LIN {X 0,Y 210.301,Z 279.738,A -85,B 0,C 180,E1 -24809.445,E2 -24809.445} C_VEL
LIN {X 0,Y 205.69,Z 270.017,A -85,B 0,C 180,E1 -24812.462,E2 -24812.462} C_VEL
LIN {X 0,Y 202.047,Z 263.223,A -85,B 0,C 180,E1 -24815.123,E2 -24815.123} C_VEL
LIN {X 0,Y 198.531,Z 257.151,A -85,B 0,C 180,E1 -24818.043,E2 -24818.043} C_VEL
LIN {X 0,Y 194.726,Z 251.083,A -85,B 0,C 180,E1 -24821.795,E2 -24821.795} C_VEL
LIN {X 0,Y 192.117,Z 247.147,A -85,B 0,C 180,E1 -24824.974,E2 -24824.974} C_VEL
LIN {X 0,Y 189.866,Z 243.661,A -85,B 0,C 180,E1 -24828.524,E2 -24828.524} C_VEL
LIN {X 0,Y 187.215,Z 239.674,A -85,B 0,C 180,E1 -24835.964,E2 -24835.964} C_VEL
LIN {X 0,Y 187.003,Z 239.077,A -85,B 0,C 180,E1 -24837.846,E2 -24837.846} C_VEL
LIN {X 0,Y 186.955,Z 239.01,A -85,B 0,C 180,E1 -24840.538,E2 -24840.538} C_VEL
LIN {X 0,Y 188.211,Z 242.32,A -85,B 0,C 180,E1 -24847.24,E2 -24847.24} C_VEL
LIN {X 0,Y 189.577,Z 244.391,A -85,B 0,C 180,E1 -24850.277,E2 -24850.277} C_VEL
LIN {X 0,Y 192.089,Z 248.48,A -85,B 0,C 180,E1 -24854.298,E2 -24854.298} C_VEL
LIN {X 0,Y 195.023,Z 253.243,A -85,B 0,C 180,E1 -24857.837,E2 -24857.837} C_VEL
LIN {X 0,Y 198.75,Z 259.543,A -85,B 0,C 180,E1 -24861.454,E2 -24861.454} C_VEL
LIN {X 0,Y 202.456,Z 266.139,A -85,B 0,C 180,E1 -24864.481,E2 -24864.481} C_VEL
LIN {X 0,Y 205.633,Z 272.337,A -85,B 0,C 180,E1 -24866.789,E2 -24866.789} C_VEL
LIN {X 0,Y 208.488,Z 283.961,A -85,B 0,C 180,E1 -24869.081,E2 -24869.081} C_VEL
LIN {X 0,Y 208.34,Z 300.022,A -85,B 0,C 180,E1 -24870.092,E2 -24870.092} C_VEL
LIN {X 0,Y 201.69,Z 376.905,A -85,B 0,C 180,E1 -24872.216,E2 -24872.216} C_VEL
LIN {X 0,Y 199.026,Z 392.933,A -85,B 0,C 180,E1 -24872.89,E2 -24872.89} C_VEL
LIN {X 0,Y 195.992,Z 405.457,A -85,B 0,C 180,E1 -24873.625,E2 -24873.625} C_VEL
LIN {X 0,Y 194.072,Z 410.997,A -85,B 0,C 180,E1 -24873.869,E2 -24873.869} C_VEL
LIN {X 0,Y 189.476,Z 419.824,A -85,B 0,C 180,E1 -24873.895,E2 -24873.895} C_VEL
LIN {X 0,Y 184.541,Z 428.454,A -85,B 0,C 180,E1 -24874.027,E2 -24874.027} C_VEL
LIN {X 0,Y 182.039,Z 433.552,A -85,B 0,C 180,E1 -24874.466,E2 -24874.466} C_VEL
LIN {X 0,Y 176.253,Z 445.926,A -85,B 0,C 180,E1 -24876.157,E2 -24876.157} C_VEL
LIN {X 0,Y 169.53,Z 458.558,A -85,B 0,C 180,E1 -24878.45,E2 -24878.45} C_VEL
LIN {X 0,Y 162.971,Z 469.426,A -85,B 0,C 180,E1 -24881.009,E2 -24881.009} C_VEL
LIN {X 0,Y 156.265,Z 479.356,A -85,B 0,C 180,E1 -24883.984,E2 -24883.984} C_VEL
LIN {X 0,Y 149.299,Z 489.115,A -85,B 0,C 180,E1 -24887.877,E2 -24887.877} C_VEL
LIN {X 0,Y 143.262,Z 496.88,A -85,B 0,C 180,E1 -24891.86,E2 -24891.86} C_VEL
LIN {X 0,Y 138.473,Z 503.139,A -85,B 0,C 180,E1 -24896.067,E2 -24896.067} C_VEL
LIN {X 0,Y 133.419,Z 509.601,A -85,B 0,C 180,E1 -24901.705,E2 -24901.705} C_VEL
LIN {X 0,Y 129.8,Z 514.638,A -85,B 0,C 180,E1 -24907.732,E2 -24907.732} C_VEL
LIN {X 0,Y 127.56,Z 518.367,A -85,B 0,C 180,E1 -24914.014,E2 -24914.014} C_VEL
LIN {X 0,Y 126.835,Z 520.883,A -85,B 0,C 180,E1 -24920.435,E2 -24920.435} C_VEL
LIN {X 0,Y 127.101,Z 521.841,A -85,B 0,C 180,E1 -24924.439,E2 -24924.439} C_VEL
LIN {X 0,Y 127.589,Z 522.401,A -85,B 0,C 180,E1 -24930.004,E2 -24930.004} C_VEL
LIN {X 0,Y 127.142,Z 521.8,A -85,B 0,C 180,E1 -24935.747,E2 -24935.747} C_VEL
LIN {X 0,Y 127.052,Z 519.741,A -85,B 0,C 180,E1 -24942.787,E2 -24942.787} C_VEL
LIN {X 0,Y 128.532,Z 516.599,A -85,B 0,C 180,E1 -24949.156,E2 -24949.156} C_VEL
LIN {X 0,Y 131.403,Z 512.192,A -85,B 0,C 180,E1 -24955.337,E2 -24955.337} C_VEL
LIN {X 0,Y 135.799,Z 506.44,A -85,B 0,C 180,E1 -24961.171,E2 -24961.171} C_VEL
LIN {X 0,Y 141.47,Z 499.175,A -85,B 0,C 180,E1 -24966.598,E2 -24966.598} C_VEL
LIN {X 0,Y 146.575,Z 492.646,A -85,B 0,C 180,E1 -24970.343,E2 -24970.343} C_VEL
LIN {X 0,Y 152.637,Z 485.303,A -85,B 0,C 180,E1 -24973.573,E2 -24973.573} C_VEL
LIN {X 0,Y 161.541,Z 483.741,A -85,B 0,C 180,E1 -24977.702,E2 -24977.702} C_VEL
LIN {X 0,Y 172.128,Z 481.337,A -85,B 0,C 180,E1 -24981.424,E2 -24981.424} C_VEL
LIN {X 0,Y 171.753,Z 480.963,A -85,B 0,C 180,E1 -24982.136,E2 -24982.136} C_VEL
LIN {X 0,Y 162.139,Z 479.16,A -85,B 0,C 180,E1 -24985.703,E2 -24985.703} C_VEL
LIN {X 0,Y 153.483,Z 476.191,A -85,B 0,C 180,E1 -24989.756,E2 -24989.756} C_VEL
LIN {X 0,Y 145.911,Z 472.001,A -85,B 0,C 180,E1 -24994.311,E2 -24994.311} C_VEL
LIN {X 0,Y 139.663,Z 466.519,A -85,B 0,C 180,E1 -24999.375,E2 -24999.375} C_VEL
LIN {X 0,Y 135.041,Z 459.696,A -85,B 0,C 180,E1 -25004.917,E2 -25004.917} C_VEL
LIN {X 0,Y 132.875,Z 454.923,A -85,B 0,C 180,E1 -25008.367,E2 -25008.367} C_VEL
LIN {X 0,Y 131.811,Z 454.489,A -85,B 0,C 180,E1 -25010.796,E2 -25010.796} C_VEL
LIN {X 0,Y 132.801,Z 449.564,A -85,B 0,C 180,E1 -25020,E2 -25020} C_VEL
LIN {X 0,Y 134.381,Z 447.309,A -85,B 0,C 180,E1 -25022.998,E2 -25022.998} C_VEL
LIN {X 0,Y 136.769,Z 444.692,A -85,B 0,C 180,E1 -25027.381,E2 -25027.381} C_VEL
LIN {X 0,Y 140.175,Z 441.466,A -85,B 0,C 180,E1 -25031.264,E2 -25031.264} C_VEL
LIN {X 0,Y 143.118,Z 439.169,A -85,B 0,C 180,E1 -25034.214,E2 -25034.214} C_VEL
LIN {X 0,Y 146.772,Z 436.106,A -85,B 0,C 180,E1 -25036.697,E2 -25036.697} C_VEL
LIN {X 0,Y 151.382,Z 432.821,A -85,B 0,C 180,E1 -25039.924,E2 -25039.924} C_VEL
LIN {X 0,Y 156.65,Z 428.519,A -85,B 0,C 180,E1 -25042.417,E2 -25042.417} C_VEL
LIN {X 0,Y 160.693,Z 425.786,A -85,B 0,C 180,E1 -25044.55,E2 -25044.55} C_VEL
LIN {X 0,Y 167.067,Z 420.351,A -85,B 0,C 180,E1 -25046.819,E2 -25046.819} C_VEL
LIN {X 0,Y 170.649,Z 417.188,A -85,B 0,C 180,E1 -25048.005,E2 -25048.005} C_VEL
LIN {X 0,Y 176.406,Z 412.41,A -85,B 0,C 180,E1 -25049.868,E2 -25049.868} C_VEL
LIN {X 0,Y 182.287,Z 406.571,A -85,B 0,C 180,E1 -25051.364,E2 -25051.364} C_VEL
LIN {X 0,Y 188.257,Z 399.411,A -85,B 0,C 180,E1 -25052.536,E2 -25052.536} C_VEL
LIN {X 0,Y 191.638,Z 395.946,A -85,B 0,C 180,E1 -25053.374,E2 -25053.374} C_VEL
LIN {X 0,Y 191.708,Z 397.569,A -85,B 0,C 180,E1 -25053.78,E2 -25053.78} C_VEL
LIN {X 0,Y 187.24,Z 410.98,A -85,B 0,C 180,E1 -25055.272,E2 -25055.272} C_VEL
LIN {X 0,Y 181.776,Z 424.211,A -85,B 0,C 180,E1 -25057.111,E2 -25057.111} C_VEL
LIN {X 0,Y 175.849,Z 436.31,A -85,B 0,C 180,E1 -25059.251,E2 -25059.251} C_VEL
LIN {X 0,Y 169.638,Z 447.434,A -85,B 0,C 180,E1 -25061.774,E2 -25061.774} C_VEL
LIN {X 0,Y 163.383,Z 457.621,A -85,B 0,C 180,E1 -25064.781,E2 -25064.781} C_VEL
LIN {X 0,Y 156.338,Z 467.581,A -85,B 0,C 180,E1 -25068.462,E2 -25068.462} C_VEL
LIN {X 0,Y 149.927,Z 475.829,A -85,B 0,C 180,E1 -25072.451,E2 -25072.451} C_VEL
LIN {X 0,Y 143.625,Z 483.517,A -85,B 0,C 180,E1 -25077.431,E2 -25077.431} C_VEL
LIN {X 0,Y 138.146,Z 489.63,A -85,B 0,C 180,E1 -25082.747,E2 -25082.747} C_VEL
LIN {X 0,Y 133.9,Z 494.331,A -85,B 0,C 180,E1 -25088.44,E2 -25088.44} C_VEL
LIN {X 0,Y 130.785,Z 497.762,A -85,B 0,C 180,E1 -25094.41,E2 -25094.41} C_VEL
LIN {X 0,Y 128.776,Z 500.015,A -85,B 0,C 180,E1 -25100.573,E2 -25100.573} C_VEL
LIN {X 0,Y 127.806,Z 501.153,A -85,B 0,C 180,E1 -25106.844,E2 -25106.844} C_VEL
LIN {X 0,Y 127.802,Z 501.162,A -85,B 0,C 180,E1 -25113.148,E2 -25113.148} C_VEL
LIN {X 0,Y 128.768,Z 500.062,A -85,B 0,C 180,E1 -25119.42,E2 -25119.42} C_VEL
LIN {X 0,Y 130.775,Z 497.85,A -85,B 0,C 180,E1 -25125.583,E2 -25125.583} C_VEL
LIN {X 0,Y 133.858,Z 494.47,A -85,B 0,C 180,E1 -25131.559,E2 -25131.559} C_VEL
LIN {X 0,Y 138.082,Z 489.818,A -85,B 0,C 180,E1 -25137.258,E2 -25137.258} C_VEL
LIN {X 0,Y 143.533,Z 483.748,A -85,B 0,C 180,E1 -25142.584,E2 -25142.584} C_VEL
LIN {X 0,Y 149.833,Z 476.111,A -85,B 0,C 180,E1 -25147.568,E2 -25147.568} C_VEL
LIN {X 0,Y 156.244,Z 467.927,A -85,B 0,C 180,E1 -25151.56,E2 -25151.56} C_VEL
LIN {X 0,Y 163.227,Z 458.042,A -85,B 0,C 180,E1 -25155.265,E2 -25155.265} C_VEL
LIN {X 0,Y 169.531,Z 447.93,A -85,B 0,C 180,E1 -25158.257,E2 -25158.257} C_VEL
LIN {X 0,Y 175.806,Z 436.902,A -85,B 0,C 180,E1 -25160.757,E2 -25160.757} C_VEL
LIN {X 0,Y 181.69,Z 424.906,A -85,B 0,C 180,E1 -25162.915,E2 -25162.915} C_VEL
LIN {X 0,Y 187.164,Z 411.807,A -85,B 0,C 180,E1 -25164.752,E2 -25164.752} C_VEL
LIN {X 0,Y 191.739,Z 398.192,A -85,B 0,C 180,E1 -25166.288,E2 -25166.288} C_VEL
LIN {X 0,Y 195.352,Z 384.362,A -85,B 0,C 180,E1 -25167.521,E2 -25167.521} C_VEL
LIN {X 0,Y 198.346,Z 369.373,A -85,B 0,C 180,E1 -25168.468,E2 -25168.468} C_VEL
LIN {X 0,Y 200.316,Z 354.638,A -85,B 0,C 180,E1 -25169.082,E2 -25169.082} C_VEL
LIN {X 0,Y 206.565,Z 283.097,A -85,B 0,C 180,E1 -25171.043,E2 -25171.043} C_VEL
LIN {X 0,Y 202.838,Z 275.011,A -85,B 0,C 180,E1 -25173.681,E2 -25173.681} C_VEL
LIN {X 0,Y 199.598,Z 268.732,A -85,B 0,C 180,E1 -25176.224,E2 -25176.224} C_VEL
LIN {X 0,Y 196.564,Z 263.306,A -85,B 0,C 180,E1 -25178.913,E2 -25178.913} C_VEL
LIN {X 0,Y 193.052,Z 257.443,A -85,B 0,C 180,E1 -25182.603,E2 -25182.603} C_VEL
LIN {X 0,Y 190.738,Z 253.83,A -85,B 0,C 180,E1 -25185.598,E2 -25185.598} C_VEL
LIN {X 0,Y 188.711,Z 250.517,A -85,B 0,C 180,E1 -25188.996,E2 -25188.996} C_VEL
LIN {X 0,Y 186.324,Z 246.732,A -85,B 0,C 180,E1 -25196.08,E2 -25196.08} C_VEL
LIN {X 0,Y 186.138,Z 246.132,A -85,B 0,C 180,E1 -25197.836,E2 -25197.836} C_VEL
LIN {X 0,Y 186.09,Z 246.061,A -85,B 0,C 180,E1 -25200.541,E2 -25200.541} C_VEL
LIN {X 0,Y 188.131,Z 250.58,A -85,B 0,C 180,E1 -25209.135,E2 -25209.135} C_VEL
LIN {X 0,Y 190.741,Z 255.196,A -85,B 0,C 180,E1 -25213.721,E2 -25213.721} C_VEL
LIN {X 0,Y 193.391,Z 259.687,A -85,B 0,C 180,E1 -25217.105,E2 -25217.105} C_VEL
LIN {X 0,Y 196.826,Z 265.796,A -85,B 0,C 180,E1 -25220.646,E2 -25220.646} C_VEL
LIN {X 0,Y 200.257,Z 272.156,A -85,B 0,C 180,E1 -25223.614,E2 -25223.614} C_VEL
LIN {X 0,Y 202.814,Z 277.371,A -85,B 0,C 180,E1 -25225.599,E2 -25225.599} C_VEL
LIN {X 0,Y 204.982,Z 286.69,A -85,B 0,C 180,E1 -25227.502,E2 -25227.502} C_VEL
LIN {X 0,Y 204.794,Z 300.471,A -85,B 0,C 180,E1 -25228.399,E2 -25228.399} C_VEL
LIN {X 0,Y 197.965,Z 376.592,A -85,B 0,C 180,E1 -25230.478,E2 -25230.478} C_VEL
LIN {X 0,Y 195.405,Z 391.525,A -85,B 0,C 180,E1 -25231.086,E2 -25231.086} C_VEL
LIN {X 0,Y 191.613,Z 406.898,A -85,B 0,C 180,E1 -25231.992,E2 -25231.992} C_VEL
LIN {X 0,Y 186.835,Z 421.579,A -85,B 0,C 180,E1 -25233.185,E2 -25233.185} C_VEL
LIN {X 0,Y 182.039,Z 433.552,A -85,B 0,C 180,E1 -25234.466,E2 -25234.466} C_VEL
LIN {X 0,Y 180.165,Z 436.986,A -85,B 0,C 180,E1 -25234.726,E2 -25234.726} C_VEL
LIN {X 0,Y 175.915,Z 442.251,A -85,B 0,C 180,E1 -25234.698,E2 -25234.698} C_VEL
LIN {X 0,Y 171.494,Z 447.391,A -85,B 0,C 180,E1 -25234.721,E2 -25234.721} C_VEL
LIN {X 0,Y 169.356,Z 450.558,A -85,B 0,C 180,E1 -25235.084,E2 -25235.084} C_VEL
LIN {X 0,Y 162.542,Z 462.474,A -85,B 0,C 180,E1 -25237.515,E2 -25237.515} C_VEL
LIN {X 0,Y 156.017,Z 472.377,A -85,B 0,C 180,E1 -25240.028,E2 -25240.028} C_VEL
LIN {X 0,Y 149.199,Z 481.767,A -85,B 0,C 180,E1 -25243.109,E2 -25243.109} C_VEL
LIN {X 0,Y 142.066,Z 491.018,A -85,B 0,C 180,E1 -25247.145,E2 -25247.145} C_VEL
LIN {X 0,Y 135.713,Z 498.723,A -85,B 0,C 180,E1 -25251.585,E2 -25251.585} C_VEL
LIN {X 0,Y 129.645,Z 505.962,A -85,B 0,C 180,E1 -25257.179,E2 -25257.179} C_VEL
LIN {X 0,Y 124.93,Z 511.693,A -85,B 0,C 180,E1 -25263.258,E2 -25263.258} C_VEL
LIN {X 0,Y 121.736,Z 516.066,A -85,B 0,C 180,E1 -25269.738,E2 -25269.738} C_VEL
LIN {X 0,Y 120.018,Z 519.18,A -85,B 0,C 180,E1 -25276.458,E2 -25276.458} C_VEL
LIN {X 0,Y 119.884,Z 521.109,A -85,B 0,C 180,E1 -25283.271,E2 -25283.271} C_VEL
LIN {X 0,Y 120.207,Z 521.624,A -85,B 0,C 180,E1 -25286.653,E2 -25286.653} C_VEL
LIN {X 0,Y 120.5,Z 521.815,A -85,B 0,C 180,E1 -25290.004,E2 -25290.004} C_VEL
LIN {X 0,Y 120.06,Z 521.279,A -85,B 0,C 180,E1 -25295.657,E2 -25295.657} C_VEL
LIN {X 0,Y 119.81,Z 520.269,A -85,B 0,C 180,E1 -25300.14,E2 -25300.14} C_VEL
LIN {X 0,Y 120.683,Z 517.725,A -85,B 0,C 180,E1 -25306.933,E2 -25306.933} C_VEL
LIN {X 0,Y 123.126,Z 513.96,A -85,B 0,C 180,E1 -25313.555,E2 -25313.555} C_VEL
LIN {X 0,Y 127.128,Z 508.897,A -85,B 0,C 180,E1 -25319.842,E2 -25319.842} C_VEL
LIN {X 0,Y 132.577,Z 502.415,A -85,B 0,C 180,E1 -25325.675,E2 -25325.675} C_VEL
LIN {X 0,Y 138.153,Z 495.656,A -85,B 0,C 180,E1 -25330.265,E2 -25330.265} C_VEL
LIN {X 0,Y 145.433,Z 487.123,A -85,B 0,C 180,E1 -25334.488,E2 -25334.488} C_VEL
LIN {X 0,Y 148.59,Z 483.626,A -85,B 0,C 180,E1 -25335.922,E2 -25335.922} C_VEL
LIN {X 0,Y 161.85,Z 481.639,A -85,B 0,C 180,E1 -25341.413,E2 -25341.413} C_VEL
LIN {X 0,Y 161.175,Z 481.066,A -85,B 0,C 180,E1 -25342.377,E2 -25342.377} C_VEL
LIN {X 0,Y 151.756,Z 478.235,A -85,B 0,C 180,E1 -25346.239,E2 -25346.239} C_VEL
LIN {X 0,Y 143.269,Z 474.219,A -85,B 0,C 180,E1 -25350.624,E2 -25350.624} C_VEL
LIN {X 0,Y 136.177,Z 468.955,A -85,B 0,C 180,E1 -25355.615,E2 -25355.615} C_VEL
LIN {X 0,Y 131.032,Z 463.521,A -85,B 0,C 180,E1 -25360.414,E2 -25360.414} C_VEL
LIN {X 0,Y 128.644,Z 462.497,A -85,B 0,C 180,E1 -25364.148,E2 -25364.148} C_VEL
LIN {X 0,Y 127.926,Z 460.868,A -85,B 0,C 180,E1 -25367.306,E2 -25367.306} C_VEL
LIN {X 0,Y 127.086,Z 459.748,A -85,B 0,C 180,E1 -25370.451,E2 -25370.451} C_VEL
LIN {X 0,Y 128.034,Z 455.043,A -85,B 0,C 180,E1 -25380,E2 -25380} C_VEL
LIN {X 0,Y 133.201,Z 449.373,A -85,B 0,C 180,E1 -25389.108,E2 -25389.108} C_VEL
LIN {X 0,Y 135.913,Z 447.051,A -85,B 0,C 180,E1 -25391.937,E2 -25391.937} C_VEL
LIN {X 0,Y 140.264,Z 443.953,A -85,B 0,C 180,E1 -25395.997,E2 -25395.997} C_VEL
LIN {X 0,Y 143.533,Z 441.403,A -85,B 0,C 180,E1 -25398.062,E2 -25398.062} C_VEL
LIN {X 0,Y 147.722,Z 438.705,A -85,B 0,C 180,E1 -25400.905,E2 -25400.905} C_VEL
LIN {X 0,Y 153.368,Z 434.562,A -85,B 0,C 180,E1 -25403.575,E2 -25403.575} C_VEL
LIN {X 0,Y 154.685,Z 433.547,A -85,B 0,C 180,E1 -25404.137,E2 -25404.137} C_VEL
LIN {X 0,Y 159.011,Z 430.838,A -85,B 0,C 180,E1 -25406.231,E2 -25406.231} C_VEL
LIN {X 0,Y 165.803,Z 425.469,A -85,B 0,C 180,E1 -25408.482,E2 -25408.482} C_VEL
LIN {X 0,Y 170.018,Z 422.026,A -85,B 0,C 180,E1 -25409.739,E2 -25409.739} C_VEL
LIN {X 0,Y 176.299,Z 417.087,A -85,B 0,C 180,E1 -25411.598,E2 -25411.598} C_VEL
LIN {X 0,Y 183.059,Z 410.79,A -85,B 0,C 180,E1 -25413.132,E2 -25413.132} C_VEL
LIN {X 0,Y 182.832,Z 412.616,A -85,B 0,C 180,E1 -25413.597,E2 -25413.597} C_VEL
LIN {X 0,Y 176.996,Z 426.093,A -85,B 0,C 180,E1 -25415.508,E2 -25415.508} C_VEL
LIN {X 0,Y 170.881,Z 438.007,A -85,B 0,C 180,E1 -25417.65,E2 -25417.65} C_VEL
LIN {X 0,Y 163.864,Z 449.871,A -85,B 0,C 180,E1 -25420.418,E2 -25420.418} C_VEL
LIN {X 0,Y 157.419,Z 459.784,A -85,B 0,C 180,E1 -25423.487,E2 -25423.487} C_VEL
LIN {X 0,Y 150.117,Z 469.477,A -85,B 0,C 180,E1 -25427.243,E2 -25427.243} C_VEL
LIN {X 0,Y 143.171,Z 477.858,A -85,B 0,C 180,E1 -25431.55,E2 -25431.55} C_VEL
LIN {X 0,Y 137.709,Z 484.102,A -85,B 0,C 180,E1 -25435.844,E2 -25435.844} C_VEL
LIN {X 0,Y 131.884,Z 490.216,A -85,B 0,C 180,E1 -25441.336,E2 -25441.336} C_VEL
LIN {X 0,Y 127.339,Z 494.916,A -85,B 0,C 180,E1 -25447.269,E2 -25447.269} C_VEL
LIN {X 0,Y 123.964,Z 498.349,A -85,B 0,C 180,E1 -25453.528,E2 -25453.528} C_VEL
LIN {X 0,Y 121.814,Z 500.599,A -85,B 0,C 180,E1 -25460.029,E2 -25460.029} C_VEL
LIN {X 0,Y 120.741,Z 501.738,A -85,B 0,C 180,E1 -25466.659,E2 -25466.659} C_VEL
LIN {X 0,Y 120.737,Z 501.747,A -85,B 0,C 180,E1 -25473.333,E2 -25473.333} C_VEL
LIN {X 0,Y 121.806,Z 500.645,A -85,B 0,C 180,E1 -25479.963,E2 -25479.963} C_VEL
LIN {X 0,Y 123.953,Z 498.436,A -85,B 0,C 180,E1 -25486.464,E2 -25486.464} C_VEL
LIN {X 0,Y 127.3,Z 495.053,A -85,B 0,C 180,E1 -25492.73,E2 -25492.73} C_VEL
LIN {X 0,Y 131.825,Z 490.401,A -85,B 0,C 180,E1 -25498.669,E2 -25498.669} C_VEL
LIN {X 0,Y 137.596,Z 484.332,A -85,B 0,C 180,E1 -25504.179,E2 -25504.179} C_VEL
LIN {X 0,Y 144.282,Z 476.693,A -85,B 0,C 180,E1 -25509.284,E2 -25509.284} C_VEL
LIN {X 0,Y 151.006,Z 468.508,A -85,B 0,C 180,E1 -25513.347,E2 -25513.347} C_VEL
LIN {X 0,Y 157.28,Z 460.181,A -85,B 0,C 180,E1 -25516.557,E2 -25516.557} C_VEL
LIN {X 0,Y 163.766,Z 450.319,A -85,B 0,C 180,E1 -25519.612,E2 -25519.612} C_VEL
LIN {X 0,Y 170.814,Z 438.546,A -85,B 0,C 180,E1 -25522.37,E2 -25522.37} C_VEL
LIN {X 0,Y 176.914,Z 426.736,A -85,B 0,C 180,E1 -25524.52,E2 -25524.52} C_VEL
LIN {X 0,Y 181.91,Z 415.45,A -85,B 0,C 180,E1 -25526.159,E2 -25526.159} C_VEL
LIN {X 0,Y 186.691,Z 402.462,A -85,B 0,C 180,E1 -25527.697,E2 -25527.697} C_VEL
LIN {X 0,Y 190.649,Z 388.919,A -85,B 0,C 180,E1 -25528.982,E2 -25528.982} C_VEL
LIN {X 0,Y 193.969,Z 374.104,A -85,B 0,C 180,E1 -25530.012,E2 -25530.012} C_VEL
LIN {X 0,Y 196.25,Z 359.84,A -85,B 0,C 180,E1 -25530.679,E2 -25530.679} C_VEL
LIN {X 0,Y 199.856,Z 320.402,A -85,B 0,C 180,E1 -25531.84,E2 -25531.84} C_VEL
LIN {X 0,Y 202.956,Z 286.419,A -85,B 0,C 180,E1 -25532.723,E2 -25532.723} C_VEL
LIN {X 0,Y 199.718,Z 279.221,A -85,B 0,C 180,E1 -25535.23,E2 -25535.23} C_VEL
LIN {X 0,Y 196.437,Z 272.696,A -85,B 0,C 180,E1 -25538.073,E2 -25538.073} C_VEL
LIN {X 0,Y 193.332,Z 267.144,A -85,B 0,C 180,E1 -25541.178,E2 -25541.178} C_VEL
LIN {X 0,Y 191.177,Z 263.47,A -85,B 0,C 180,E1 -25543.721,E2 -25543.721} C_VEL
LIN {X 0,Y 189.421,Z 260.538,A -85,B 0,C 180,E1 -25546.181,E2 -25546.181} C_VEL
LIN {X 0,Y 187.57,Z 257.366,A -85,B 0,C 180,E1 -25549.475,E2 -25549.475} C_VEL
LIN {X 0,Y 185.347,Z 253.38,A -85,B 0,C 180,E1 -25557.011,E2 -25557.011} C_VEL
LIN {X 0,Y 185.223,Z 253.121,A -85,B 0,C 180,E1 -25560.543,E2 -25560.543} C_VEL
LIN {X 0,Y 187.07,Z 257.557,A -85,B 0,C 180,E1 -25568.779,E2 -25568.779} C_VEL
LIN {X 0,Y 189.332,Z 261.737,A -85,B 0,C 180,E1 -25573.005,E2 -25573.005} C_VEL
LIN {X 0,Y 191.838,Z 266.266,A -85,B 0,C 180,E1 -25576.426,E2 -25576.426} C_VEL
LIN {X 0,Y 194.952,Z 272.062,A -85,B 0,C 180,E1 -25579.831,E2 -25579.831} C_VEL
LIN {X 0,Y 198.041,Z 278.053,A -85,B 0,C 180,E1 -25582.673,E2 -25582.673} C_VEL
LIN {X 0,Y 200.081,Z 282.443,A -85,B 0,C 180,E1 -25584.376,E2 -25584.376} C_VEL
LIN {X 0,Y 201.578,Z 289.429,A -85,B 0,C 180,E1 -25585.837,E2 -25585.837} C_VEL
LIN {X 0,Y 201.377,Z 301.467,A -85,B 0,C 180,E1 -25586.658,E2 -25586.658} C_VEL
LIN {X 0,Y 194.542,Z 375.348,A -85,B 0,C 180,E1 -25588.648,E2 -25588.648} C_VEL
LIN {X 0,Y 192.015,Z 390.106,A -85,B 0,C 180,E1 -25589.231,E2 -25589.231} C_VEL
LIN {X 0,Y 188.294,Z 405.073,A -85,B 0,C 180,E1 -25590.071,E2 -25590.071} C_VEL
LIN {X 0,Y 183.734,Z 419.063,A -85,B 0,C 180,E1 -25591.151,E2 -25591.151} C_VEL
LIN {X 0,Y 178.2,Z 432.753,A -85,B 0,C 180,E1 -25592.547,E2 -25592.547} C_VEL
LIN {X 0,Y 172.136,Z 445.352,A -85,B 0,C 180,E1 -25594.238,E2 -25594.238} C_VEL
LIN {X 0,Y 169.356,Z 450.558,A -85,B 0,C 180,E1 -25595.084,E2 -25595.084} C_VEL
LIN {X 0,Y 166.353,Z 455.267,A -85,B 0,C 180,E1 -25595.783,E2 -25595.783} C_VEL
LIN {X 0,Y 160.083,Z 462.596,A -85,B 0,C 180,E1 -25596.579,E2 -25596.579} C_VEL
LIN {X 0,Y 153.536,Z 469.587,A -85,B 0,C 180,E1 -25597.532,E2 -25597.532} C_VEL
LIN {X 0,Y 150.13,Z 473.642,A -85,B 0,C 180,E1 -25598.509,E2 -25598.509} C_VEL
LIN {X 0,Y 143.287,Z 482.598,A -85,B 0,C 180,E1 -25601.59,E2 -25601.59} C_VEL
LIN {X 0,Y 135.88,Z 491.624,A -85,B 0,C 180,E1 -25605.719,E2 -25605.719} C_VEL
LIN {X 0,Y 130.108,Z 498.128,A -85,B 0,C 180,E1 -25609.6,E2 -25609.6} C_VEL
LIN {X 0,Y 123.647,Z 505.369,A -85,B 0,C 180,E1 -25615.367,E2 -25615.367} C_VEL
LIN {X 0,Y 118.533,Z 511.099,A -85,B 0,C 180,E1 -25621.689,E2 -25621.689} C_VEL
LIN {X 0,Y 114.999,Z 515.471,A -85,B 0,C 180,E1 -25628.494,E2 -25628.494} C_VEL
LIN {X 0,Y 113.05,Z 518.587,A -85,B 0,C 180,E1 -25635.606,E2 -25635.606} C_VEL
LIN {X 0,Y 112.761,Z 520.516,A -85,B 0,C 180,E1 -25642.844,E2 -25642.844} C_VEL
LIN {X 0,Y 113.097,Z 521.035,A -85,B 0,C 180,E1 -25646.442,E2 -25646.442} C_VEL
LIN {X 0,Y 113.414,Z 521.229,A -85,B 0,C 180,E1 -25650.005,E2 -25650.005} C_VEL
LIN {X 0,Y 112.988,Z 520.752,A -85,B 0,C 180,E1 -25655.605,E2 -25655.605} C_VEL
LIN {X 0,Y 112.735,Z 519.674,A -85,B 0,C 180,E1 -25660.784,E2 -25660.784} C_VEL
LIN {X 0,Y 113.822,Z 517.131,A -85,B 0,C 180,E1 -25667.987,E2 -25667.987} C_VEL
LIN {X 0,Y 116.86,Z 512.975,A -85,B 0,C 180,E1 -25675.565,E2 -25675.565} C_VEL
LIN {X 0,Y 120.938,Z 508.302,A -85,B 0,C 180,E1 -25681.539,E2 -25681.539} C_VEL
LIN {X 0,Y 126.797,Z 501.82,A -85,B 0,C 180,E1 -25687.572,E2 -25687.572} C_VEL
LIN {X 0,Y 132.195,Z 495.676,A -85,B 0,C 180,E1 -25691.902,E2 -25691.902} C_VEL
LIN {X 0,Y 139.29,Z 487.783,A -85,B 0,C 180,E1 -25695.976,E2 -25695.976} C_VEL
LIN {X 0,Y 144.835,Z 481.78,A -85,B 0,C 180,E1 -25698.385,E2 -25698.385} C_VEL
LIN {X 0,Y 152.452,Z 481.01,A -85,B 0,C 180,E1 -25701.605,E2 -25701.605} C_VEL
LIN {X 0,Y 150.629,Z 480.237,A -85,B 0,C 180,E1 -25702.66,E2 -25702.66} C_VEL
LIN {X 0,Y 141.375,Z 476.387,A -85,B 0,C 180,E1 -25706.851,E2 -25706.851} C_VEL
LIN {X 0,Y 132.785,Z 471.077,A -85,B 0,C 180,E1 -25711.983,E2 -25711.983} C_VEL
LIN {X 0,Y 129.929,Z 470.653,A -85,B 0,C 180,E1 -25714.36,E2 -25714.36} C_VEL
LIN {X 0,Y 127.417,Z 469.706,A -85,B 0,C 180,E1 -25717.288,E2 -25717.288} C_VEL
LIN {X 0,Y 125.607,Z 468.411,A -85,B 0,C 180,E1 -25720.384,E2 -25720.384} C_VEL
LIN {X 0,Y 123.763,Z 467.51,A -85,B 0,C 180,E1 -25723.505,E2 -25723.505} C_VEL
LIN {X 0,Y 121.853,Z 463.487,A -85,B 0,C 180,E1 -25733.376,E2 -25733.376} C_VEL
LIN {X 0,Y 124.383,Z 458.597,A -85,B 0,C 180,E1 -25743.239,E2 -25743.239} C_VEL
LIN {X 0,Y 129.591,Z 453.901,A -85,B 0,C 180,E1 -25750.942,E2 -25750.942} C_VEL
LIN {X 0,Y 137.376,Z 448.579,A -85,B 0,C 180,E1 -25757.876,E2 -25757.876} C_VEL
LIN {X 0,Y 141.415,Z 445.794,A -85,B 0,C 180,E1 -25760.358,E2 -25760.358} C_VEL
LIN {X 0,Y 145.362,Z 443.456,A -85,B 0,C 180,E1 -25762.755,E2 -25762.755} C_VEL
LIN {X 0,Y 152.686,Z 438.453,A -85,B 0,C 180,E1 -25765.931,E2 -25765.931} C_VEL
LIN {X 0,Y 157.305,Z 435.762,A -85,B 0,C 180,E1 -25767.977,E2 -25767.977} C_VEL
LIN {X 0,Y 165.891,Z 429.376,A -85,B 0,C 180,E1 -25770.556,E2 -25770.556} C_VEL
LIN {X 0,Y 173.688,Z 423.665,A -85,B 0,C 180,E1 -25772.732,E2 -25772.732} C_VEL
LIN {X 0,Y 173.834,Z 424.87,A -85,B 0,C 180,E1 -25773.311,E2 -25773.311} C_VEL
LIN {X 0,Y 167.888,Z 436.324,A -85,B 0,C 180,E1 -25775.28,E2 -25775.28} C_VEL
LIN {X 0,Y 161.342,Z 447.312,A -85,B 0,C 180,E1 -25777.675,E2 -25777.675} C_VEL
LIN {X 0,Y 154.802,Z 457.211,A -85,B 0,C 180,E1 -25780.492,E2 -25780.492} C_VEL
LIN {X 0,Y 148.163,Z 466.117,A -85,B 0,C 180,E1 -25783.662,E2 -25783.662} C_VEL
LIN {X 0,Y 140.912,Z 474.831,A -85,B 0,C 180,E1 -25787.672,E2 -25787.672} C_VEL
LIN {X 0,Y 133.526,Z 482.945,A -85,B 0,C 180,E1 -25792.746,E2 -25792.746} C_VEL
LIN {X 0,Y 127.119,Z 489.43,A -85,B 0,C 180,E1 -25798.312,E2 -25798.312} C_VEL
LIN {X 0,Y 121.948,Z 494.478,A -85,B 0,C 180,E1 -25804.386,E2 -25804.386} C_VEL
LIN {X 0,Y 118.857,Z 497.371,A -85,B 0,C 180,E1 -25809.216,E2 -25809.216} C_VEL
LIN {X 0,Y 115.849,Z 500.239,A -85,B 0,C 180,E1 -25816.084,E2 -25816.084} C_VEL
LIN {X 0,Y 114.098,Z 501.891,A -85,B 0,C 180,E1 -25822.919,E2 -25822.919} C_VEL
LIN {X 0,Y 113.553,Z 502.47,A -85,B 0,C 180,E1 -25829.995,E2 -25829.995} C_VEL
LIN {X 0,Y 114.09,Z 501.919,A -85,B 0,C 180,E1 -25837.072,E2 -25837.072} C_VEL
LIN {X 0,Y 115.873,Z 500.265,A -85,B 0,C 180,E1 -25844.036,E2 -25844.036} C_VEL
LIN {X 0,Y 118.803,Z 497.483,A -85,B 0,C 180,E1 -25850.785,E2 -25850.785} C_VEL
LIN {X 0,Y 123.067,Z 493.478,A -85,B 0,C 180,E1 -25857.179,E2 -25857.179} C_VEL
LIN {X 0,Y 128.516,Z 488.142,A -85,B 0,C 180,E1 -25863.146,E2 -25863.146} C_VEL
LIN {X 0,Y 133.434,Z 483.168,A -85,B 0,C 180,E1 -25867.275,E2 -25867.275} C_VEL
LIN {X 0,Y 139.827,Z 476.192,A -85,B 0,C 180,E1 -25871.752,E2 -25871.752} C_VEL
LIN {X 0,Y 146.984,Z 467.773,A -85,B 0,C 180,E1 -25875.82,E2 -25875.82} C_VEL
LIN {X 0,Y 153.566,Z 459.2,A -85,B 0,C 180,E1 -25879.031,E2 -25879.031} C_VEL
LIN {X 0,Y 160.443,Z 449.082,A -85,B 0,C 180,E1 -25882.036,E2 -25882.036} C_VEL
LIN {X 0,Y 167.826,Z 436.905,A -85,B 0,C 180,E1 -25884.739,E2 -25884.739} C_VEL
LIN {X 0,Y 174.151,Z 424.678,A -85,B 0,C 180,E1 -25886.858,E2 -25886.858} C_VEL
LIN {X 0,Y 180.019,Z 411.257,A -85,B 0,C 180,E1 -25888.644,E2 -25888.644} C_VEL
LIN {X 0,Y 184.599,Z 398.158,A -85,B 0,C 180,E1 -25890.077,E2 -25890.077} C_VEL
LIN {X 0,Y 188.413,Z 384.452,A -85,B 0,C 180,E1 -25891.223,E2 -25891.223} C_VEL
LIN {X 0,Y 191.564,Z 369.159,A -85,B 0,C 180,E1 -25892.145,E2 -25892.145} C_VEL
LIN {X 0,Y 193.669,Z 353.253,A -85,B 0,C 180,E1 -25892.762,E2 -25892.762} C_VEL
LIN {X 0,Y 199.546,Z 289.853,A -85,B 0,C 180,E1 -25894.44,E2 -25894.44} C_VEL
LIN {X 0,Y 196.111,Z 282.184,A -85,B 0,C 180,E1 -25897.394,E2 -25897.394} C_VEL
LIN {X 0,Y 192.871,Z 275.752,A -85,B 0,C 180,E1 -25900.603,E2 -25900.603} C_VEL
LIN {X 0,Y 190.002,Z 270.502,A -85,B 0,C 180,E1 -25904.019,E2 -25904.019} C_VEL
LIN {X 0,Y 188.042,Z 267.118,A -85,B 0,C 180,E1 -25906.904,E2 -25906.904} C_VEL
LIN {X 0,Y 186.402,Z 264.187,A -85,B 0,C 180,E1 -25910.04,E2 -25910.04} C_VEL
LIN {X 0,Y 184.497,Z 260.648,A -85,B 0,C 180,E1 -25916.724,E2 -25916.724} C_VEL
LIN {X 0,Y 184.405,Z 260.253,A -85,B 0,C 180,E1 -25917.816,E2 -25917.816} C_VEL
LIN {X 0,Y 184.353,Z 260.144,A -85,B 0,C 180,E1 -25920.409,E2 -25920.409} C_VEL
LIN {X 0,Y 186.019,Z 264.504,A -85,B 0,C 180,E1 -25928.418,E2 -25928.418} C_VEL
LIN {X 0,Y 188.027,Z 268.466,A -85,B 0,C 180,E1 -25932.411,E2 -25932.411} C_VEL
LIN {X 0,Y 190.317,Z 272.816,A -85,B 0,C 180,E1 -25935.735,E2 -25935.735} C_VEL
LIN {X 0,Y 193.062,Z 278.231,A -85,B 0,C 180,E1 -25938.943,E2 -25938.943} C_VEL
LIN {X 0,Y 195.802,Z 283.789,A -85,B 0,C 180,E1 -25941.642,E2 -25941.642} C_VEL
LIN {X 0,Y 197.501,Z 287.764,A -85,B 0,C 180,E1 -25943.182,E2 -25943.182} C_VEL
LIN {X 0,Y 198.415,Z 292.417,A -85,B 0,C 180,E1 -25944.177,E2 -25944.177} C_VEL
LIN {X 0,Y 198.232,Z 301.619,A -85,B 0,C 180,E1 -25944.836,E2 -25944.836} C_VEL
LIN {X 0,Y 191.293,Z 374.305,A -85,B 0,C 180,E1 -25946.756,E2 -25946.756} C_VEL
LIN {X 0,Y 188.841,Z 388.688,A -85,B 0,C 180,E1 -25947.316,E2 -25947.316} C_VEL
LIN {X 0,Y 185.193,Z 403.249,A -85,B 0,C 180,E1 -25948.082,E2 -25948.082} C_VEL
LIN {X 0,Y 180.863,Z 416.541,A -85,B 0,C 180,E1 -25949.044,E2 -25949.044} C_VEL
LIN {X 0,Y 175.18,Z 430.616,A -85,B 0,C 180,E1 -25950.403,E2 -25950.403} C_VEL
LIN {X 0,Y 168.226,Z 444.777,A -85,B 0,C 180,E1 -25952.229,E2 -25952.229} C_VEL
LIN {X 0,Y 161.556,Z 456.478,A -85,B 0,C 180,E1 -25954.262,E2 -25954.262} C_VEL
LIN {X 0,Y 155.237,Z 466.477,A -85,B 0,C 180,E1 -25956.532,E2 -25956.532} C_VEL
LIN {X 0,Y 150.13,Z 473.642,A -85,B 0,C 180,E1 -25958.509,E2 -25958.509} C_VEL
LIN {X 0,Y 146.682,Z 477.612,A -85,B 0,C 180,E1 -25959.58,E2 -25959.58} C_VEL
LIN {X 0,Y 139.775,Z 483.682,A -85,B 0,C 180,E1 -25961.059,E2 -25961.059} C_VEL
LIN {X 0,Y 132.834,Z 489.343,A -85,B 0,C 180,E1 -25962.828,E2 -25962.828} C_VEL
LIN {X 0,Y 129.412,Z 492.558,A -85,B 0,C 180,E1 -25964.372,E2 -25964.372} C_VEL
LIN {X 0,Y 122.878,Z 499.505,A -85,B 0,C 180,E1 -25968.878,E2 -25968.878} C_VEL
LIN {X 0,Y 116.259,Z 506.349,A -85,B 0,C 180,E1 -25974.956,E2 -25974.956} C_VEL
LIN {X 0,Y 110.995,Z 511.852,A -85,B 0,C 180,E1 -25981.859,E2 -25981.859} C_VEL
LIN {X 0,Y 108.33,Z 514.877,A -85,B 0,C 180,E1 -25987.097,E2 -25987.097} C_VEL
LIN {X 0,Y 106.102,Z 517.993,A -85,B 0,C 180,E1 -25994.641,E2 -25994.641} C_VEL
LIN {X 0,Y 105.661,Z 519.924,A -85,B 0,C 180,E1 -26002.36,E2 -26002.36} C_VEL
LIN {X 0,Y 105.991,Z 520.447,A -85,B 0,C 180,E1 -26006.203,E2 -26006.203} C_VEL
LIN {X 0,Y 106.327,Z 520.644,A -85,B 0,C 180,E1 -26010.005,E2 -26010.005} C_VEL
LIN {X 0,Y 105.905,Z 520.232,A -85,B 0,C 180,E1 -26015.491,E2 -26015.491} C_VEL
LIN {X 0,Y 105.698,Z 519.081,A -85,B 0,C 180,E1 -26021.511,E2 -26021.511} C_VEL
LIN {X 0,Y 107.009,Z 516.536,A -85,B 0,C 180,E1 -26029.176,E2 -26029.176} C_VEL
LIN {X 0,Y 110.168,Z 512.656,A -85,B 0,C 180,E1 -26036.734,E2 -26036.734} C_VEL
LIN {X 0,Y 114.847,Z 507.706,A -85,B 0,C 180,E1 -26043.424,E2 -26043.424} C_VEL
LIN {X 0,Y 121.141,Z 501.222,A -85,B 0,C 180,E1 -26049.66,E2 -26049.66} C_VEL
LIN {X 0,Y 127.078,Z 494.947,A -85,B 0,C 180,E1 -26054.153,E2 -26054.153} C_VEL
LIN {X 0,Y 134.444,Z 487.197,A -85,B 0,C 180,E1 -26058.156,E2 -26058.156} C_VEL
LIN {X 0,Y 141.378,Z 479.792,A -85,B 0,C 180,E1 -26060.967,E2 -26060.967} C_VEL
LIN {X 0,Y 141.968,Z 479.757,A -85,B 0,C 180,E1 -26061.237,E2 -26061.237} C_VEL
LIN {X 0,Y 141.74,Z 479.12,A -85,B 0,C 180,E1 -26062.303,E2 -26062.303} C_VEL
LIN {X 0,Y 138.072,Z 477.581,A -85,B 0,C 180,E1 -26063.947,E2 -26063.947} C_VEL
LIN {X 0,Y 131.623,Z 476.96,A -85,B 0,C 180,E1 -26067.728,E2 -26067.728} C_VEL
LIN {X 0,Y 128.442,Z 475.964,A -85,B 0,C 180,E1 -26070.498,E2 -26070.498} C_VEL
LIN {X 0,Y 125.167,Z 475.351,A -85,B 0,C 180,E1 -26073.309,E2 -26073.309} C_VEL
LIN {X 0,Y 121.648,Z 474.015,A -85,B 0,C 180,E1 -26077.584,E2 -26077.584} C_VEL
LIN {X 0,Y 118.714,Z 472.303,A -85,B 0,C 180,E1 -26082.783,E2 -26082.783} C_VEL
LIN {X 0,Y 116.606,Z 468.447,A -85,B 0,C 180,E1 -26093.077,E2 -26093.077} C_VEL
LIN {X 0,Y 119.147,Z 463.793,A -85,B 0,C 180,E1 -26103.382,E2 -26103.382} C_VEL
LIN {X 0,Y 126.755,Z 457.737,A -85,B 0,C 180,E1 -26113.674,E2 -26113.674} C_VEL
LIN {X 0,Y 132.51,Z 454.231,A -85,B 0,C 180,E1 -26118.556,E2 -26118.556} C_VEL
LIN {X 0,Y 139.499,Z 449.978,A -85,B 0,C 180,E1 -26122.79,E2 -26122.79} C_VEL
LIN {X 0,Y 143.017,Z 448.044,A -85,B 0,C 180,E1 -26124.69,E2 -26124.69} C_VEL
LIN {X 0,Y 151.403,Z 442.827,A -85,B 0,C 180,E1 -26128.114,E2 -26128.114} C_VEL
LIN {X 0,Y 155.604,Z 440.536,A -85,B 0,C 180,E1 -26129.791,E2 -26129.791} C_VEL
LIN {X 0,Y 164.118,Z 434.676,A -85,B 0,C 180,E1 -26132.184,E2 -26132.184} C_VEL
LIN {X 0,Y 165.245,Z 433.857,A -85,B 0,C 180,E1 -26132.449,E2 -26132.449} C_VEL
LIN {X 0,Y 165.267,Z 434.608,A -85,B 0,C 180,E1 -26132.869,E2 -26132.869} C_VEL
LIN {X 0,Y 158.811,Z 445.335,A -85,B 0,C 180,E1 -26135.016,E2 -26135.016} C_VEL
LIN {X 0,Y 151.462,Z 456.213,A -85,B 0,C 180,E1 -26137.92,E2 -26137.92} C_VEL
LIN {X 0,Y 144.557,Z 465.307,A -85,B 0,C 180,E1 -26141.095,E2 -26141.095} C_VEL
LIN {X 0,Y 136.816,Z 474.25,A -85,B 0,C 180,E1 -26145.06,E2 -26145.06} C_VEL
LIN {X 0,Y 129.776,Z 481.65,A -85,B 0,C 180,E1 -26149.464,E2 -26149.464} C_VEL
LIN {X 0,Y 124.46,Z 486.958,A -85,B 0,C 180,E1 -26153.631,E2 -26153.631} C_VEL
LIN {X 0,Y 118.203,Z 492.71,A -85,B 0,C 180,E1 -26159.638,E2 -26159.638} C_VEL
LIN {X 0,Y 114.407,Z 496.087,A -85,B 0,C 180,E1 -26164.527,E2 -26164.527} C_VEL
LIN {X 0,Y 110.456,Z 499.52,A -85,B 0,C 180,E1 -26171.445,E2 -26171.445} C_VEL
LIN {X 0,Y 107.931,Z 501.767,A -85,B 0,C 180,E1 -26178.73,E2 -26178.73} C_VEL
LIN {X 0,Y 106.621,Z 502.907,A -85,B 0,C 180,E1 -26186.216,E2 -26186.216} C_VEL
LIN {X 0,Y 106.618,Z 502.916,A -85,B 0,C 180,E1 -26193.775,E2 -26193.775} C_VEL
LIN {X 0,Y 107.923,Z 501.812,A -85,B 0,C 180,E1 -26201.261,E2 -26201.261} C_VEL
LIN {X 0,Y 110.443,Z 499.605,A -85,B 0,C 180,E1 -26208.547,E2 -26208.547} C_VEL
LIN {X 0,Y 114.35,Z 496.223,A -85,B 0,C 180,E1 -26215.476,E2 -26215.476} C_VEL
LIN {X 0,Y 119.547,Z 491.572,A -85,B 0,C 180,E1 -26221.939,E2 -26221.939} C_VEL
LIN {X 0,Y 126.092,Z 485.501,A -85,B 0,C 180,E1 -26227.809,E2 -26227.809} C_VEL
LIN {X 0,Y 133.622,Z 477.855,A -85,B 0,C 180,E1 -26233.132,E2 -26233.132} C_VEL
LIN {X 0,Y 141.038,Z 469.668,A -85,B 0,C 180,E1 -26237.301,E2 -26237.301} C_VEL
LIN {X 0,Y 147.888,Z 461.339,A -85,B 0,C 180,E1 -26240.549,E2 -26240.549} C_VEL
LIN {X 0,Y 154.89,Z 451.573,A -85,B 0,C 180,E1 -26243.578,E2 -26243.578} C_VEL
LIN {X 0,Y 161.914,Z 440.735,A -85,B 0,C 180,E1 -26246.106,E2 -26246.106} C_VEL
LIN {X 0,Y 168.442,Z 429.131,A -85,B 0,C 180,E1 -26248.218,E2 -26248.218} C_VEL
LIN {X 0,Y 173.763,Z 418.117,A -85,B 0,C 180,E1 -26249.822,E2 -26249.822} C_VEL
LIN {X 0,Y 179.426,Z 403.879,A -85,B 0,C 180,E1 -26251.485,E2 -26251.485} C_VEL
LIN {X 0,Y 183.771,Z 390.01,A -85,B 0,C 180,E1 -26252.757,E2 -26252.757} C_VEL
LIN {X 0,Y 187.306,Z 375.158,A -85,B 0,C 180,E1 -26253.758,E2 -26253.758} C_VEL
LIN {X 0,Y 189.85,Z 359.667,A -85,B 0,C 180,E1 -26254.454,E2 -26254.454} C_VEL
LIN {X 0,Y 196.277,Z 293.316,A -85,B 0,C 180,E1 -26256.245,E2 -26256.245} C_VEL
LIN {X 0,Y 193.653,Z 287.353,A -85,B 0,C 180,E1 -26258.72,E2 -26258.72} C_VEL
LIN {X 0,Y 190.926,Z 281.631,A -85,B 0,C 180,E1 -26261.664,E2 -26261.664} C_VEL
LIN {X 0,Y 188.432,Z 276.908,A -85,B 0,C 180,E1 -26264.866,E2 -26264.866} C_VEL
LIN {X 0,Y 186.769,Z 273.825,A -85,B 0,C 180,E1 -26267.504,E2 -26267.504} C_VEL
LIN {X 0,Y 185.391,Z 271.161,A -85,B 0,C 180,E1 -26270.306,E2 -26270.306} C_VEL
LIN {X 0,Y 183.626,Z 267.755,A -85,B 0,C 180,E1 -26276.709,E2 -26276.709} C_VEL
LIN {X 0,Y 183.538,Z 267.318,A -85,B 0,C 180,E1 -26277.805,E2 -26277.805} C_VEL
LIN {X 0,Y 183.481,Z 267.251,A -85,B 0,C 180,E1 -26280.411,E2 -26280.411} C_VEL
LIN {X 0,Y 184.978,Z 271.438,A -85,B 0,C 180,E1 -26288.054,E2 -26288.054} C_VEL
LIN {X 0,Y 186.742,Z 275.19,A -85,B 0,C 180,E1 -26291.808,E2 -26291.808} C_VEL
LIN {X 0,Y 188.871,Z 279.46,A -85,B 0,C 180,E1 -26295.098,E2 -26295.098} C_VEL
LIN {X 0,Y 191.299,Z 284.567,A -85,B 0,C 180,E1 -26298.128,E2 -26298.128} C_VEL
LIN {X 0,Y 193.689,Z 289.676,A -85,B 0,C 180,E1 -26300.649,E2 -26300.649} C_VEL
LIN {X 0,Y 194.964,Z 292.75,A -85,B 0,C 180,E1 -26301.892,E2 -26301.892} C_VEL
LIN {X 0,Y 195.419,Z 295.822,A -85,B 0,C 180,E1 -26302.5,E2 -26302.5} C_VEL
LIN {X 0,Y 195.102,Z 303.763,A -85,B 0,C 180,E1 -26303.009,E2 -26303.009} C_VEL
LIN {X 0,Y 188.107,Z 374.572,A -85,B 0,C 180,E1 -26304.846,E2 -26304.846} C_VEL
LIN {X 0,Y 185.31,Z 389.933,A -85,B 0,C 180,E1 -26305.438,E2 -26305.438} C_VEL
LIN {X 0,Y 181.216,Z 405.245,A -85,B 0,C 180,E1 -26306.261,E2 -26306.261} C_VEL
LIN {X 0,Y 176.069,Z 419.892,A -85,B 0,C 180,E1 -26307.367,E2 -26307.367} C_VEL
LIN {X 0,Y 170.245,Z 433.184,A -85,B 0,C 180,E1 -26308.697,E2 -26308.697} C_VEL
LIN {X 0,Y 163.139,Z 446.77,A -85,B 0,C 180,E1 -26310.511,E2 -26310.511} C_VEL
LIN {X 0,Y 156.364,Z 457.946,A -85,B 0,C 180,E1 -26312.525,E2 -26312.525} C_VEL
LIN {X 0,Y 149.774,Z 467.68,A -85,B 0,C 180,E1 -26314.804,E2 -26314.804} C_VEL
LIN {X 0,Y 142.21,Z 477.604,A -85,B 0,C 180,E1 -26317.754,E2 -26317.754} C_VEL
LIN {X 0,Y 134.059,Z 487.345,A -85,B 0,C 180,E1 -26321.671,E2 -26321.671} C_VEL
LIN {X 0,Y 129.412,Z 492.558,A -85,B 0,C 180,E1 -26324.372,E2 -26324.372} C_VEL
LIN {X 0,Y 126.015,Z 495.666,A -85,B 0,C 180,E1 -26326.05,E2 -26326.05} C_VEL
LIN {X 0,Y 119.141,Z 500.282,A -85,B 0,C 180,E1 -26328.605,E2 -26328.605} C_VEL
LIN {X 0,Y 112.429,Z 504.436,A -85,B 0,C 180,E1 -26331.582,E2 -26331.582} C_VEL
LIN {X 0,Y 109.399,Z 506.725,A -85,B 0,C 180,E1 -26333.912,E2 -26333.912} C_VEL
LIN {X 0,Y 103.688,Z 512.26,A -85,B 0,C 180,E1 -26341.682,E2 -26341.682} C_VEL
LIN {X 0,Y 100.217,Z 515.992,A -85,B 0,C 180,E1 -26349.479,E2 -26349.479} C_VEL
LIN {X 0,Y 98.634,Z 518.512,A -85,B 0,C 180,E1 -26357.663,E2 -26357.663} C_VEL
LIN {X 0,Y 98.897,Z 519.859,A -85,B 0,C 180,E1 -26365.93,E2 -26365.93} C_VEL
LIN {X 0,Y 99.24,Z 520.058,A -85,B 0,C 180,E1 -26370.005,E2 -26370.005} C_VEL
LIN {X 0,Y 98.826,Z 519.71,A -85,B 0,C 180,E1 -26375.377,E2 -26375.377} C_VEL
LIN {X 0,Y 98.661,Z 518.487,A -85,B 0,C 180,E1 -26382.345,E2 -26382.345} C_VEL
LIN {X 0,Y 100.225,Z 515.94,A -85,B 0,C 180,E1 -26390.53,E2 -26390.53} C_VEL
LIN {X 0,Y 103.673,Z 512.173,A -85,B 0,C 180,E1 -26398.334,E2 -26398.334} C_VEL
LIN {X 0,Y 108.902,Z 507.11,A -85,B 0,C 180,E1 -26405.513,E2 -26405.513} C_VEL
LIN {X 0,Y 115.667,Z 500.625,A -85,B 0,C 180,E1 -26411.947,E2 -26411.947} C_VEL
LIN {X 0,Y 122.82,Z 493.565,A -85,B 0,C 180,E1 -26416.968,E2 -26416.968} C_VEL
LIN {X 0,Y 131.07,Z 485.364,A -85,B 0,C 180,E1 -26421.037,E2 -26421.037} C_VEL
LIN {X 0,Y 133.66,Z 482.661,A -85,B 0,C 180,E1 -26422.072,E2 -26422.072} C_VEL
LIN {X 0,Y 131.088,Z 481.926,A -85,B 0,C 180,E1 -26423.862,E2 -26423.862} C_VEL
LIN {X 0,Y 126.99,Z 481.42,A -85,B 0,C 180,E1 -26426.398,E2 -26426.398} C_VEL
LIN {X 0,Y 123.646,Z 480.48,A -85,B 0,C 180,E1 -26429.233,E2 -26429.233} C_VEL
LIN {X 0,Y 117.478,Z 478.987,A -85,B 0,C 180,E1 -26435.244,E2 -26435.244} C_VEL
LIN {X 0,Y 112.26,Z 475.67,A -85,B 0,C 180,E1 -26445.498,E2 -26445.498} C_VEL
LIN {X 0,Y 111.471,Z 471.784,A -85,B 0,C 180,E1 -26456.386,E2 -26456.386} C_VEL
LIN {X 0,Y 115.619,Z 467.045,A -85,B 0,C 180,E1 -26466.983,E2 -26466.983} C_VEL
LIN {X 0,Y 127.48,Z 459.602,A -85,B 0,C 180,E1 -26479.317,E2 -26479.317} C_VEL
LIN {X 0,Y 140.675,Z 452.464,A -85,B 0,C 180,E1 -26486.721,E2 -26486.721} C_VEL
LIN {X 0,Y 148.475,Z 447.925,A -85,B 0,C 180,E1 -26489.658,E2 -26489.658} C_VEL
LIN {X 0,Y 153.888,Z 445.154,A -85,B 0,C 180,E1 -26491.682,E2 -26491.682} C_VEL
LIN {X 0,Y 155.366,Z 444.232,A -85,B 0,C 180,E1 -26492.108,E2 -26492.108} C_VEL
LIN {X 0,Y 154.827,Z 445.961,A -85,B 0,C 180,E1 -26492.882,E2 -26492.882} C_VEL
LIN {X 0,Y 147.209,Z 456.797,A -85,B 0,C 180,E1 -26495.742,E2 -26495.742} C_VEL
LIN {X 0,Y 140.006,Z 465.89,A -85,B 0,C 180,E1 -26498.911,E2 -26498.911} C_VEL
LIN {X 0,Y 131.905,Z 474.833,A -85,B 0,C 180,E1 -26502.889,E2 -26502.889} C_VEL
LIN {X 0,Y 124.474,Z 482.235,A -85,B 0,C 180,E1 -26507.343,E2 -26507.343} C_VEL
LIN {X 0,Y 118.834,Z 487.543,A -85,B 0,C 180,E1 -26511.607,E2 -26511.607} C_VEL
LIN {X 0,Y 112.136,Z 493.297,A -85,B 0,C 180,E1 -26517.805,E2 -26517.805} C_VEL
LIN {X 0,Y 108.039,Z 496.675,A -85,B 0,C 180,E1 -26522.907,E2 -26522.907} C_VEL
LIN {X 0,Y 103.777,Z 500.105,A -85,B 0,C 180,E1 -26530.203,E2 -26530.203} C_VEL
LIN {X 0,Y 101.013,Z 502.351,A -85,B 0,C 180,E1 -26537.947,E2 -26537.947} C_VEL
LIN {X 0,Y 99.568,Z 503.491,A -85,B 0,C 180,E1 -26545.947,E2 -26545.947} C_VEL
LIN {X 0,Y 99.564,Z 503.5,A -85,B 0,C 180,E1 -26554.043,E2 -26554.043} C_VEL
LIN {X 0,Y 101.006,Z 502.395,A -85,B 0,C 180,E1 -26562.043,E2 -26562.043} C_VEL
LIN {X 0,Y 103.764,Z 500.188,A -85,B 0,C 180,E1 -26569.789,E2 -26569.789} C_VEL
LIN {X 0,Y 107.982,Z 496.808,A -85,B 0,C 180,E1 -26577.097,E2 -26577.097} C_VEL
LIN {X 0,Y 113.579,Z 492.157,A -85,B 0,C 180,E1 -26583.836,E2 -26583.836} C_VEL
LIN {X 0,Y 120.559,Z 486.085,A -85,B 0,C 180,E1 -26589.879,E2 -26589.879} C_VEL
LIN {X 0,Y 128.532,Z 478.437,A -85,B 0,C 180,E1 -26595.296,E2 -26595.296} C_VEL
LIN {X 0,Y 136.342,Z 470.247,A -85,B 0,C 180,E1 -26599.486,E2 -26599.486} C_VEL
LIN {X 0,Y 143.474,Z 461.92,A -85,B 0,C 180,E1 -26602.743,E2 -26602.743} C_VEL
LIN {X 0,Y 150.752,Z 452.21,A -85,B 0,C 180,E1 -26605.724,E2 -26605.724} C_VEL
LIN {X 0,Y 158.087,Z 441.307,A -85,B 0,C 180,E1 -26608.23,E2 -26608.23} C_VEL
LIN {X 0,Y 164.831,Z 429.701,A -85,B 0,C 180,E1 -26610.305,E2 -26610.305} C_VEL
LIN {X 0,Y 170.322,Z 418.681,A -85,B 0,C 180,E1 -26611.877,E2 -26611.877} C_VEL
LIN {X 0,Y 176.107,Z 404.593,A -85,B 0,C 180,E1 -26613.489,E2 -26613.489} C_VEL
LIN {X 0,Y 180.379,Z 391.5,A -85,B 0,C 180,E1 -26614.685,E2 -26614.685} C_VEL
LIN {X 0,Y 184.054,Z 376.904,A -85,B 0,C 180,E1 -26615.661,E2 -26615.661} C_VEL
LIN {X 0,Y 186.666,Z 362.354,A -85,B 0,C 180,E1 -26616.315,E2 -26616.315} C_VEL
LIN {X 0,Y 189.385,Z 335.855,A -85,B 0,C 180,E1 -26617.103,E2 -26617.103} C_VEL
LIN {X 0,Y 193.197,Z 297.017,A -85,B 0,C 180,E1 -26618.094,E2 -26618.094} C_VEL
LIN {X 0,Y 190.748,Z 291.208,A -85,B 0,C 180,E1 -26620.704,E2 -26620.704} C_VEL
LIN {X 0,Y 188.277,Z 286.033,A -85,B 0,C 180,E1 -26623.742,E2 -26623.742} C_VEL
LIN {X 0,Y 186.265,Z 281.952,A -85,B 0,C 180,E1 -26626.78,E2 -26626.78} C_VEL
LIN {X 0,Y 184.226,Z 277.925,A -85,B 0,C 180,E1 -26630.946,E2 -26630.946} C_VEL
LIN {X 0,Y 182.727,Z 274.749,A -85,B 0,C 180,E1 -26636.968,E2 -26636.968} C_VEL
LIN {X 0,Y 182.67,Z 274.397,A -85,B 0,C 180,E1 -26637.795,E2 -26637.795} C_VEL
LIN {X 0,Y 182.609,Z 274.349,A -85,B 0,C 180,E1 -26640.413,E2 -26640.413} C_VEL
LIN {X 0,Y 183.942,Z 278.392,A -85,B 0,C 180,E1 -26647.685,E2 -26647.685} C_VEL
LIN {X 0,Y 185.481,Z 281.896,A -85,B 0,C 180,E1 -26651.197,E2 -26651.197} C_VEL
LIN {X 0,Y 187.404,Z 286.002,A -85,B 0,C 180,E1 -26654.386,E2 -26654.386} C_VEL
LIN {X 0,Y 189.705,Z 291.145,A -85,B 0,C 180,E1 -26657.448,E2 -26657.448} C_VEL
LIN {X 0,Y 192.224,Z 296.968,A -85,B 0,C 180,E1 -26660.254,E2 -26660.254} C_VEL
LIN {X 0,Y 192.609,Z 298.4,A -85,B 0,C 180,E1 -26660.701,E2 -26660.701} C_VEL
LIN {X 0,Y 192.3,Z 304.581,A -85,B 0,C 180,E1 -26661.085,E2 -26661.085} C_VEL
LIN {X 0,Y 185.273,Z 373.769,A -85,B 0,C 180,E1 -26662.842,E2 -26662.842} C_VEL
LIN {X 0,Y 182.559,Z 388.515,A -85,B 0,C 180,E1 -26663.385,E2 -26663.385} C_VEL
LIN {X 0,Y 178.562,Z 403.423,A -85,B 0,C 180,E1 -26664.136,E2 -26664.136} C_VEL
LIN {X 0,Y 173.65,Z 417.378,A -85,B 0,C 180,E1 -26665.108,E2 -26665.108} C_VEL
LIN {X 0,Y 167.685,Z 431.048,A -85,B 0,C 180,E1 -26666.388,E2 -26666.388} C_VEL
LIN {X 0,Y 161.089,Z 443.631,A -85,B 0,C 180,E1 -26667.945,E2 -26667.945} C_VEL
LIN {X 0,Y 153.963,Z 455.319,A -85,B 0,C 180,E1 -26669.861,E2 -26669.861} C_VEL
LIN {X 0,Y 145.824,Z 467.099,A -85,B 0,C 180,E1 -26672.505,E2 -26672.505} C_VEL
LIN {X 0,Y 137.936,Z 477.018,A -85,B 0,C 180,E1 -26675.398,E2 -26675.398} C_VEL
LIN {X 0,Y 130.571,Z 485.507,A -85,B 0,C 180,E1 -26678.704,E2 -26678.704} C_VEL
LIN {X 0,Y 121.73,Z 494.775,A -85,B 0,C 180,E1 -26683.673,E2 -26683.673} C_VEL
LIN {X 0,Y 113.857,Z 502.53,A -85,B 0,C 180,E1 -26689.606,E2 -26689.606} C_VEL
LIN {X 0,Y 109.399,Z 506.725,A -85,B 0,C 180,E1 -26693.912,E2 -26693.912} C_VEL
LIN {X 0,Y 106.539,Z 508.876,A -85,B 0,C 180,E1 -26696.412,E2 -26696.412} C_VEL
LIN {X 0,Y 100.644,Z 511.886,A -85,B 0,C 180,E1 -26700.498,E2 -26700.498} C_VEL
LIN {X 0,Y 96.182,Z 513.887,A -85,B 0,C 180,E1 -26704.151,E2 -26704.151} C_VEL
LIN {X 0,Y 93.808,Z 515.185,A -85,B 0,C 180,E1 -26707.328,E2 -26707.328} C_VEL
LIN {X 0,Y 93.327,Z 515.576,A -85,B 0,C 180,E1 -26708.474,E2 -26708.474} C_VEL
LIN {X 0,Y 91.64,Z 517.919,A -85,B 0,C 180,E1 -26716.704,E2 -26716.704} C_VEL
LIN {X 0,Y 91.77,Z 519.269,A -85,B 0,C 180,E1 -26725.613,E2 -26725.613} C_VEL
LIN {X 0,Y 92.153,Z 519.472,A -85,B 0,C 180,E1 -26730.006,E2 -26730.006} C_VEL
LIN {X 0,Y 91.751,Z 519.186,A -85,B 0,C 180,E1 -26735.266,E2 -26735.266} C_VEL
LIN {X 0,Y 91.664,Z 517.893,A -85,B 0,C 180,E1 -26743.304,E2 -26743.304} C_VEL
LIN {X 0,Y 93.515,Z 515.345,A -85,B 0,C 180,E1 -26752.077,E2 -26752.077} C_VEL
LIN {X 0,Y 97.381,Z 511.576,A -85,B 0,C 180,E1 -26760.35,E2 -26760.35} C_VEL
LIN {X 0,Y 103.132,Z 506.515,A -85,B 0,C 180,E1 -26767.835,E2 -26767.835} C_VEL
LIN {X 0,Y 110.401,Z 500.028,A -85,B 0,C 180,E1 -26774.453,E2 -26774.453} C_VEL
LIN {X 0,Y 117.823,Z 493.192,A -85,B 0,C 180,E1 -26779.385,E2 -26779.385} C_VEL
LIN {X 0,Y 124.101,Z 487.258,A -85,B 0,C 180,E1 -26782.457,E2 -26782.457} C_VEL
LIN {X 0,Y 124.678,Z 485.944,A -85,B 0,C 180,E1 -26783.429,E2 -26783.429} C_VEL
LIN {X 0,Y 122.292,Z 485.649,A -85,B 0,C 180,E1 -26784.923,E2 -26784.923} C_VEL
LIN {X 0,Y 112.343,Z 483.272,A -85,B 0,C 180,E1 -26794.03,E2 -26794.03} C_VEL
LIN {X 0,Y 106.739,Z 480.083,A -85,B 0,C 180,E1 -26804.73,E2 -26804.73} C_VEL
LIN {X 0,Y 105.832,Z 476.338,A -85,B 0,C 180,E1 -26816.193,E2 -26816.193} C_VEL
LIN {X 0,Y 110.034,Z 471.819,A -85,B 0,C 180,E1 -26827.34,E2 -26827.34} C_VEL
LIN {X 0,Y 122.311,Z 464.684,A -85,B 0,C 180,E1 -26840.168,E2 -26840.168} C_VEL
LIN {X 0,Y 128.708,Z 461.427,A -85,B 0,C 180,E1 -26844.176,E2 -26844.176} C_VEL
LIN {X 0,Y 137.817,Z 456.986,A -85,B 0,C 180,E1 -26848.642,E2 -26848.642} C_VEL
LIN {X 0,Y 146.778,Z 452.236,A -85,B 0,C 180,E1 -26851.783,E2 -26851.783} C_VEL
LIN {X 0,Y 146.231,Z 453.335,A -85,B 0,C 180,E1 -26852.3,E2 -26852.3} C_VEL
LIN {X 0,Y 139.438,Z 462.117,A -85,B 0,C 180,E1 -26855.006,E2 -26855.006} C_VEL
LIN {X 0,Y 130.74,Z 471.813,A -85,B 0,C 180,E1 -26858.784,E2 -26858.784} C_VEL
LIN {X 0,Y 122.604,Z 479.841,A -85,B 0,C 180,E1 -26863.037,E2 -26863.037} C_VEL
LIN {X 0,Y 115.321,Z 486.448,A -85,B 0,C 180,E1 -26867.899,E2 -26867.899} C_VEL
LIN {X 0,Y 107.828,Z 492.564,A -85,B 0,C 180,E1 -26874.078,E2 -26874.078} C_VEL
LIN {X 0,Y 101.773,Z 497.261,A -85,B 0,C 180,E1 -26881.088,E2 -26881.088} C_VEL
LIN {X 0,Y 97.135,Z 500.691,A -85,B 0,C 180,E1 -26888.786,E2 -26888.786} C_VEL
LIN {X 0,Y 94.117,Z 502.935,A -85,B 0,C 180,E1 -26897.049,E2 -26897.049} C_VEL
LIN {X 0,Y 92.518,Z 504.076,A -85,B 0,C 180,E1 -26905.638,E2 -26905.638} C_VEL
LIN {X 0,Y 92.515,Z 504.084,A -85,B 0,C 180,E1 -26914.351,E2 -26914.351} C_VEL
LIN {X 0,Y 94.11,Z 502.978,A -85,B 0,C 180,E1 -26922.94,E2 -26922.94} C_VEL
LIN {X 0,Y 97.119,Z 500.774,A -85,B 0,C 180,E1 -26931.206,E2 -26931.206} C_VEL
LIN {X 0,Y 101.718,Z 497.393,A -85,B 0,C 180,E1 -26938.918,E2 -26938.918} C_VEL
LIN {X 0,Y 107.752,Z 492.742,A -85,B 0,C 180,E1 -26945.939,E2 -26945.939} C_VEL
LIN {X 0,Y 115.204,Z 486.668,A -85,B 0,C 180,E1 -26952.142,E2 -26952.142} C_VEL
LIN {X 0,Y 122.522,Z 480.105,A -85,B 0,C 180,E1 -26956.992,E2 -26956.992} C_VEL
LIN {X 0,Y 130.654,Z 472.12,A -85,B 0,C 180,E1 -26961.251,E2 -26961.251} C_VEL
LIN {X 0,Y 139.295,Z 462.499,A -85,B 0,C 180,E1 -26965.066,E2 -26965.066} C_VEL
LIN {X 0,Y 147.407,Z 452.096,A -85,B 0,C 180,E1 -26968.193,E2 -26968.193} C_VEL
LIN {X 0,Y 155.852,Z 439.763,A -85,B 0,C 180,E1 -26970.884,E2 -26970.884} C_VEL
LIN {X 0,Y 162.831,Z 427.749,A -85,B 0,C 180,E1 -26972.891,E2 -26972.891} C_VEL
LIN {X 0,Y 169.244,Z 414.624,A -85,B 0,C 180,E1 -26974.572,E2 -26974.572} C_VEL
LIN {X 0,Y 174.683,Z 400.724,A -85,B 0,C 180,E1 -26976.023,E2 -26976.023} C_VEL
LIN {X 0,Y 179.166,Z 386.083,A -85,B 0,C 180,E1 -26977.181,E2 -26977.181} C_VEL
LIN {X 0,Y 182.62,Z 370.77,A -85,B 0,C 180,E1 -26978.027,E2 -26978.027} C_VEL
LIN {X 0,Y 184.883,Z 355.145,A -85,B 0,C 180,E1 -26978.593,E2 -26978.593} C_VEL
LIN {X 0,Y 190.327,Z 300.714,A -85,B 0,C 180,E1 -26980,E2 -26980} C_VEL
LIN {X 0,Y 187.679,Z 294.465,A -85,B 0,C 180,E1 -26983.234,E2 -26983.234} C_VEL
LIN {X 0,Y 185.44,Z 289.652,A -85,B 0,C 180,E1 -26986.584,E2 -26986.584} C_VEL
LIN {X 0,Y 184.092,Z 286.829,A -85,B 0,C 180,E1 -26989.135,E2 -26989.135} C_VEL
LIN {X 0,Y 183.138,Z 284.791,A -85,B 0,C 180,E1 -26991.448,E2 -26991.448} C_VEL
LIN {X 0,Y 181.855,Z 281.86,A -85,B 0,C 180,E1 -26996.954,E2 -26996.954} C_VEL
LIN {X 0,Y 181.742,Z 281.35,A -85,B 0,C 180,E1 -26998.892,E2 -26998.892} C_VEL
LIN {X 0,Y 181.733,Z 281.433,A -85,B 0,C 180,E1 -27000.277,E2 -27000.277} C_VEL
LIN {X 0,Y 182.87,Z 285.218,A -85,B 0,C 180,E1 -27007.175,E2 -27007.175} C_VEL
LIN {X 0,Y 184.306,Z 288.762,A -85,B 0,C 180,E1 -27010.713,E2 -27010.713} C_VEL
LIN {X 0,Y 185.924,Z 292.456,A -85,B 0,C 180,E1 -27013.596,E2 -27013.596} C_VEL
LIN {X 0,Y 188.001,Z 297.433,A -85,B 0,C 180,E1 -27016.584,E2 -27016.584} C_VEL
LIN {X 0,Y 189.9,Z 302.11,A -85,B 0,C 180,E1 -27018.895,E2 -27018.895} C_VEL
LIN {X 0,Y 189.805,Z 304.66,A -85,B 0,C 180,E1 -27019.097,E2 -27019.097} C_VEL
LIN {X 0,Y 182.624,Z 373.356,A -85,B 0,C 180,E1 -27020.791,E2 -27020.791} C_VEL
LIN {X 0,Y 179.666,Z 388.871,A -85,B 0,C 180,E1 -27021.343,E2 -27021.343} C_VEL
LIN {X 0,Y 175.384,Z 404.141,A -85,B 0,C 180,E1 -27022.088,E2 -27022.088} C_VEL
LIN {X 0,Y 169.986,Z 418.764,A -85,B 0,C 180,E1 -27023.095,E2 -27023.095} C_VEL
LIN {X 0,Y 163.893,Z 432.048,A -85,B 0,C 180,E1 -27024.332,E2 -27024.332} C_VEL
LIN {X 0,Y 156.373,Z 445.618,A -85,B 0,C 180,E1 -27025.998,E2 -27025.998} C_VEL
LIN {X 0,Y 149.221,Z 456.684,A -85,B 0,C 180,E1 -27027.862,E2 -27027.862} C_VEL
LIN {X 0,Y 142.122,Z 466.519,A -85,B 0,C 180,E1 -27030.082,E2 -27030.082} C_VEL
LIN {X 0,Y 133.912,Z 476.432,A -85,B 0,C 180,E1 -27032.898,E2 -27032.898} C_VEL
LIN {X 0,Y 124.971,Z 486.167,A -85,B 0,C 180,E1 -27036.746,E2 -27036.746} C_VEL
LIN {X 0,Y 116.536,Z 494.511,A -85,B 0,C 180,E1 -27041.345,E2 -27041.345} C_VEL
LIN {X 0,Y 108.459,Z 501.935,A -85,B 0,C 180,E1 -27047.133,E2 -27047.133} C_VEL
LIN {X 0,Y 101.505,Z 508.029,A -85,B 0,C 180,E1 -27053.954,E2 -27053.954} C_VEL
LIN {X 0,Y 96.899,Z 512.129,A -85,B 0,C 180,E1 -27060.498,E2 -27060.498} C_VEL
LIN {X 0,Y 93.327,Z 515.576,A -85,B 0,C 180,E1 -27068.474,E2 -27068.474} C_VEL
LIN {X 0,Y 91.727,Z 516.704,A -85,B 0,C 180,E1 -27071.937,E2 -27071.937} C_VEL
LIN {X 0,Y 88.094,Z 517.935,A -85,B 0,C 180,E1 -27077.759,E2 -27077.759} C_VEL
LIN {X 0,Y 85.607,Z 518.509,A -85,B 0,C 180,E1 -27082.747,E2 -27082.747} C_VEL
LIN {X 0,Y 84.793,Z 518.757,A -85,B 0,C 180,E1 -27086.71,E2 -27086.71} C_VEL
LIN {X 0,Y 84.829,Z 518.801,A -85,B 0,C 180,E1 -27088.05,E2 -27088.05} C_VEL
LIN {X 0,Y 85.064,Z 518.886,A -85,B 0,C 180,E1 -27090.006,E2 -27090.006} C_VEL
LIN {X 0,Y 84.673,Z 518.655,A -85,B 0,C 180,E1 -27095.117,E2 -27095.117} C_VEL
LIN {X 0,Y 84.676,Z 517.298,A -85,B 0,C 180,E1 -27104.424,E2 -27104.424} C_VEL
LIN {X 0,Y 86.892,Z 514.75,A -85,B 0,C 180,E1 -27113.86,E2 -27113.86} C_VEL
LIN {X 0,Y 91.246,Z 510.981,A -85,B 0,C 180,E1 -27122.633,E2 -27122.633} C_VEL
LIN {X 0,Y 97.54,Z 505.919,A -85,B 0,C 180,E1 -27130.433,E2 -27130.433} C_VEL
LIN {X 0,Y 105.373,Z 499.432,A -85,B 0,C 180,E1 -27137.201,E2 -27137.201} C_VEL
LIN {X 0,Y 113.427,Z 492.491,A -85,B 0,C 180,E1 -27142.19,E2 -27142.19} C_VEL
LIN {X 0,Y 115.848,Z 490.32,A -85,B 0,C 180,E1 -27143.393,E2 -27143.393} C_VEL
LIN {X 0,Y 115.384,Z 489.166,A -85,B 0,C 180,E1 -27144.948,E2 -27144.948} C_VEL
LIN {X 0,Y 107.108,Z 487.325,A -85,B 0,C 180,E1 -27152.658,E2 -27152.658} C_VEL
LIN {X 0,Y 101.07,Z 484.255,A -85,B 0,C 180,E1 -27163.851,E2 -27163.851} C_VEL
LIN {X 0,Y 99.971,Z 480.68,A -85,B 0,C 180,E1 -27175.969,E2 -27175.969} C_VEL
LIN {X 0,Y 104.257,Z 476.35,A -85,B 0,C 180,E1 -27187.749,E2 -27187.749} C_VEL
LIN {X 0,Y 116.984,Z 469.513,A -85,B 0,C 180,E1 -27201.129,E2 -27201.129} C_VEL
LIN {X 0,Y 125.412,Z 465.623,A -85,B 0,C 180,E1 -27206.273,E2 -27206.273} C_VEL
LIN {X 0,Y 137.126,Z 460.279,A -85,B 0,C 180,E1 -27211.451,E2 -27211.451} C_VEL
LIN {X 0,Y 136.767,Z 461.126,A -85,B 0,C 180,E1 -27212.012,E2 -27212.012} C_VEL
LIN {X 0,Y 128.962,Z 469.766,A -85,B 0,C 180,E1 -27215.163,E2 -27215.163} C_VEL
LIN {X 0,Y 120.261,Z 478.254,A -85,B 0,C 180,E1 -27219.25,E2 -27219.25} C_VEL
LIN {X 0,Y 111.688,Z 485.755,A -85,B 0,C 180,E1 -27224.33,E2 -27224.33} C_VEL
LIN {X 0,Y 104.051,Z 491.775,A -85,B 0,C 180,E1 -27230.078,E2 -27230.078} C_VEL
LIN {X 0,Y 97.12,Z 496.826,A -85,B 0,C 180,E1 -27237.124,E2 -27237.124} C_VEL
LIN {X 0,Y 92.896,Z 499.715,A -85,B 0,C 180,E1 -27242.998,E2 -27242.998} C_VEL
LIN {X 0,Y 88.647,Z 502.545,A -85,B 0,C 180,E1 -27251.505,E2 -27251.505} C_VEL
LIN {X 0,Y 86.13,Z 504.227,A -85,B 0,C 180,E1 -27260.602,E2 -27260.602} C_VEL
LIN {X 0,Y 85.273,Z 504.808,A -85,B 0,C 180,E1 -27269.994,E2 -27269.994} C_VEL
LIN {X 0,Y 86.122,Z 504.253,A -85,B 0,C 180,E1 -27279.387,E2 -27279.387} C_VEL
LIN {X 0,Y 88.641,Z 502.606,A -85,B 0,C 180,E1 -27288.484,E2 -27288.484} C_VEL
LIN {X 0,Y 92.85,Z 499.821,A -85,B 0,C 180,E1 -27297.004,E2 -27297.004} C_VEL
LIN {X 0,Y 98.655,Z 495.819,A -85,B 0,C 180,E1 -27304.737,E2 -27304.737} C_VEL
LIN {X 0,Y 105.946,Z 490.472,A -85,B 0,C 180,E1 -27311.549,E2 -27311.549} C_VEL
LIN {X 0,Y 114.368,Z 483.642,A -85,B 0,C 180,E1 -27317.504,E2 -27317.504} C_VEL
LIN {X 0,Y 122.622,Z 476.292,A -85,B 0,C 180,E1 -27321.998,E2 -27321.998} C_VEL
LIN {X 0,Y 131.495,Z 467.409,A -85,B 0,C 180,E1 -27325.93,E2 -27325.93} C_VEL
LIN {X 0,Y 139.328,Z 458.346,A -85,B 0,C 180,E1 -27329.031,E2 -27329.031} C_VEL
LIN {X 0,Y 147.543,Z 447.584,A -85,B 0,C 180,E1 -27331.779,E2 -27331.779} C_VEL
LIN {X 0,Y 155.431,Z 435.754,A -85,B 0,C 180,E1 -27333.975,E2 -27333.975} C_VEL
LIN {X 0,Y 161.908,Z 424.168,A -85,B 0,C 180,E1 -27335.712,E2 -27335.712} C_VEL
LIN {X 0,Y 168.383,Z 410.402,A -85,B 0,C 180,E1 -27337.279,E2 -27337.279} C_VEL
LIN {X 0,Y 173.616,Z 396.292,A -85,B 0,C 180,E1 -27338.588,E2 -27338.588} C_VEL
LIN {X 0,Y 177.679,Z 382.177,A -85,B 0,C 180,E1 -27339.555,E2 -27339.555} C_VEL
LIN {X 0,Y 180.873,Z 366.7,A -85,B 0,C 180,E1 -27340.303,E2 -27340.303} C_VEL
LIN {X 0,Y 183.028,Z 349.57,A -85,B 0,C 180,E1 -27340.835,E2 -27340.835} C_VEL
LIN {X 0,Y 187.641,Z 304.764,A -85,B 0,C 180,E1 -27341.948,E2 -27341.948} C_VEL
LIN {X 0,Y 185.62,Z 299.68,A -85,B 0,C 180,E1 -27344.771,E2 -27344.771} C_VEL
LIN {X 0,Y 183.403,Z 294.563,A -85,B 0,C 180,E1 -27348.674,E2 -27348.674} C_VEL
LIN {X 0,Y 182.065,Z 291.644,A -85,B 0,C 180,E1 -27351.956,E2 -27351.956} C_VEL
LIN {X 0,Y 180.928,Z 288.592,A -85,B 0,C 180,E1 -27357.774,E2 -27357.774} C_VEL
LIN {X 0,Y 180.857,Z 288.622,A -85,B 0,C 180,E1 -27360.417,E2 -27360.417} C_VEL
LIN {X 0,Y 181.854,Z 292.154,A -85,B 0,C 180,E1 -27366.797,E2 -27366.797} C_VEL
LIN {X 0,Y 183.08,Z 295.487,A -85,B 0,C 180,E1 -27370.087,E2 -27370.087} C_VEL
LIN {X 0,Y 184.479,Z 298.913,A -85,B 0,C 180,E1 -27372.793,E2 -27372.793} C_VEL
LIN {X 0,Y 186.358,Z 303.744,A -85,B 0,C 180,E1 -27375.727,E2 -27375.727} C_VEL
LIN {X 0,Y 187.356,Z 306.331,A -85,B 0,C 180,E1 -27377.074,E2 -27377.074} C_VEL
LIN {X 0,Y 180.399,Z 371.471,A -85,B 0,C 180,E1 -27378.63,E2 -27378.63} C_VEL
LIN {X 0,Y 177.602,Z 386.567,A -85,B 0,C 180,E1 -27379.141,E2 -27379.141} C_VEL
LIN {X 0,Y 173.635,Z 401.051,A -85,B 0,C 180,E1 -27379.779,E2 -27379.779} C_VEL
LIN {X 0,Y 168.893,Z 414.299,A -85,B 0,C 180,E1 -27380.575,E2 -27380.575} C_VEL
LIN {X 0,Y 162.631,Z 428.342,A -85,B 0,C 180,E1 -27381.713,E2 -27381.713} C_VEL
LIN {X 0,Y 155.696,Z 441.2,A -85,B 0,C 180,E1 -27383.126,E2 -27383.126} C_VEL
LIN {X 0,Y 148.088,Z 453.089,A -85,B 0,C 180,E1 -27384.828,E2 -27384.828} C_VEL
LIN {X 0,Y 140.126,Z 464.152,A -85,B 0,C 180,E1 -27387.104,E2 -27387.104} C_VEL
LIN {X 0,Y 131.566,Z 474.349,A -85,B 0,C 180,E1 -27389.777,E2 -27389.777} C_VEL
LIN {X 0,Y 122.1,Z 484.33,A -85,B 0,C 180,E1 -27393.433,E2 -27393.433} C_VEL
LIN {X 0,Y 113.22,Z 492.772,A -85,B 0,C 180,E1 -27397.833,E2 -27397.833} C_VEL
LIN {X 0,Y 105.349,Z 499.577,A -85,B 0,C 180,E1 -27402.8,E2 -27402.8} C_VEL
LIN {X 0,Y 97.518,Z 506.039,A -85,B 0,C 180,E1 -27409.57,E2 -27409.57} C_VEL
LIN {X 0,Y 91.267,Z 511.073,A -85,B 0,C 180,E1 -27417.389,E2 -27417.389} C_VEL
LIN {X 0,Y 86.891,Z 514.805,A -85,B 0,C 180,E1 -27426.152,E2 -27426.152} C_VEL
LIN {X 0,Y 84.655,Z 517.325,A -85,B 0,C 180,E1 -27435.585,E2 -27435.585} C_VEL
LIN {X 0,Y 84.667,Z 518.68,A -85,B 0,C 180,E1 -27445.245,E2 -27445.245} C_VEL
LIN {X 0,Y 84.829,Z 518.801,A -85,B 0,C 180,E1 -27448.05,E2 -27448.05} C_VEL
LIN {X 0,Y 84.652,Z 518.833,A -85,B 0,C 180,E1 -27450.676,E2 -27450.676} C_VEL
LIN {X 0,Y 83.839,Z 518.681,A -85,B 0,C 180,E1 -27453.274,E2 -27453.274} C_VEL
LIN {X 0,Y 81.274,Z 518.039,A -85,B 0,C 180,E1 -27458.479,E2 -27458.479} C_VEL
LIN {X 0,Y 78.834,Z 517.064,A -85,B 0,C 180,E1 -27464.038,E2 -27464.038} C_VEL
LIN {X 0,Y 78.251,Z 516.176,A -85,B 0,C 180,E1 -27468.412,E2 -27468.412} C_VEL
LIN {X 0,Y 78.456,Z 515.808,A -85,B 0,C 180,E1 -27469.87,E2 -27469.87} C_VEL
LIN {X 0,Y 82.542,Z 512.426,A -85,B 0,C 180,E1 -27480.728,E2 -27480.728} C_VEL
LIN {X 0,Y 88.496,Z 508.023,A -85,B 0,C 180,E1 -27489.451,E2 -27489.451} C_VEL
LIN {X 0,Y 96.241,Z 502.27,A -85,B 0,C 180,E1 -27496.914,E2 -27496.914} C_VEL
LIN {X 0,Y 105.376,Z 495.012,A -85,B 0,C 180,E1 -27503.17,E2 -27503.17} C_VEL
LIN {X 0,Y 107.549,Z 493.237,A -85,B 0,C 180,E1 -27504.349,E2 -27504.349} C_VEL
LIN {X 0,Y 106.93,Z 492.232,A -85,B 0,C 180,E1 -27506.064,E2 -27506.064} C_VEL
LIN {X 0,Y 101.797,Z 491.121,A -85,B 0,C 180,E1 -27511.101,E2 -27511.101} C_VEL
LIN {X 0,Y 94.834,Z 487.737,A -85,B 0,C 180,E1 -27524.471,E2 -27524.471} C_VEL
LIN {X 0,Y 94.83,Z 483.463,A -85,B 0,C 180,E1 -27540,E2 -27540} C_VEL
LIN {X 0,Y 104.007,Z 477.495,A -85,B 0,C 180,E1 -27555.682,E2 -27555.682} C_VEL
LIN {X 0,Y 117.361,Z 471.638,A -85,B 0,C 180,E1 -27566.062,E2 -27566.062} C_VEL
LIN {X 0,Y 127.276,Z 467.471,A -85,B 0,C 180,E1 -27570.831,E2 -27570.831} C_VEL
LIN {X 0,Y 126.656,Z 468.77,A -85,B 0,C 180,E1 -27571.899,E2 -27571.899} C_VEL
LIN {X 0,Y 117.197,Z 477.751,A -85,B 0,C 180,E1 -27575.941,E2 -27575.941} C_VEL
LIN {X 0,Y 108.318,Z 485.207,A -85,B 0,C 180,E1 -27580.674,E2 -27580.674} C_VEL
LIN {X 0,Y 100.83,Z 490.863,A -85,B 0,C 180,E1 -27585.806,E2 -27585.806} C_VEL
LIN {X 0,Y 92.977,Z 496.251,A -85,B 0,C 180,E1 -27592.786,E2 -27592.786} C_VEL
LIN {X 0,Y 86.649,Z 500.3,A -85,B 0,C 180,E1 -27600.873,E2 -27600.873} C_VEL
LIN {X 0,Y 81.953,Z 503.131,A -85,B 0,C 180,E1 -27609.932,E2 -27609.932} C_VEL
LIN {X 0,Y 79.173,Z 504.811,A -85,B 0,C 180,E1 -27619.767,E2 -27619.767} C_VEL
LIN {X 0,Y 78.207,Z 505.392,A -85,B 0,C 180,E1 -27629.993,E2 -27629.993} C_VEL
LIN {X 0,Y 79.166,Z 504.836,A -85,B 0,C 180,E1 -27640.221,E2 -27640.221} C_VEL
LIN {X 0,Y 81.945,Z 503.191,A -85,B 0,C 180,E1 -27650.056,E2 -27650.056} C_VEL
LIN {X 0,Y 86.583,Z 500.407,A -85,B 0,C 180,E1 -27659.138,E2 -27659.138} C_VEL
LIN {X 0,Y 92.919,Z 496.403,A -85,B 0,C 180,E1 -27667.228,E2 -27667.228} C_VEL
LIN {X 0,Y 100.758,Z 491.055,A -85,B 0,C 180,E1 -27674.22,E2 -27674.22} C_VEL
LIN {X 0,Y 109.705,Z 484.224,A -85,B 0,C 180,E1 -27680.234,E2 -27680.234} C_VEL
LIN {X 0,Y 118.401,Z 476.871,A -85,B 0,C 180,E1 -27684.694,E2 -27684.694} C_VEL
LIN {X 0,Y 127.664,Z 467.988,A -85,B 0,C 180,E1 -27688.562,E2 -27688.562} C_VEL
LIN {X 0,Y 135.821,Z 458.924,A -85,B 0,C 180,E1 -27691.592,E2 -27691.592} C_VEL
LIN {X 0,Y 145.062,Z 447.196,A -85,B 0,C 180,E1 -27694.457,E2 -27694.457} C_VEL
LIN {X 0,Y 153.206,Z 435.17,A -85,B 0,C 180,E1 -27696.548,E2 -27696.548} C_VEL
LIN {X 0,Y 159.895,Z 423.342,A -85,B 0,C 180,E1 -27698.196,E2 -27698.196} C_VEL
LIN {X 0,Y 166.358,Z 409.651,A -85,B 0,C 180,E1 -27699.663,E2 -27699.663} C_VEL
LIN {X 0,Y 171.91,Z 394.664,A -85,B 0,C 180,E1 -27700.965,E2 -27700.965} C_VEL
LIN {X 0,Y 176.067,Z 379.853,A -85,B 0,C 180,E1 -27701.887,E2 -27701.887} C_VEL
LIN {X 0,Y 179.151,Z 364.196,A -85,B 0,C 180,E1 -27702.525,E2 -27702.525} C_VEL
LIN {X 0,Y 181.961,Z 339.296,A -85,B 0,C 180,E1 -27703.212,E2 -27703.212} C_VEL
LIN {X 0,Y 185.158,Z 308.816,A -85,B 0,C 180,E1 -27703.973,E2 -27703.973} C_VEL
LIN {X 0,Y 183.184,Z 303.725,A -85,B 0,C 180,E1 -27707.255,E2 -27707.255} C_VEL
LIN {X 0,Y 181.672,Z 300.102,A -85,B 0,C 180,E1 -27710.537,E2 -27710.537} C_VEL
LIN {X 0,Y 181.007,Z 298.491,A -85,B 0,C 180,E1 -27712.47,E2 -27712.47} C_VEL
LIN {X 0,Y 180.053,Z 295.729,A -85,B 0,C 180,E1 -27717.763,E2 -27717.763} C_VEL
LIN {X 0,Y 179.985,Z 295.649,A -85,B 0,C 180,E1 -27720.209,E2 -27720.209} C_VEL
LIN {X 0,Y 180.844,Z 299.113,A -85,B 0,C 180,E1 -27726.415,E2 -27726.415} C_VEL
LIN {X 0,Y 181.878,Z 302.199,A -85,B 0,C 180,E1 -27729.452,E2 -27729.452} C_VEL
LIN {X 0,Y 183.178,Z 305.664,A -85,B 0,C 180,E1 -27732.182,E2 -27732.182} C_VEL
LIN {X 0,Y 184.806,Z 310.208,A -85,B 0,C 180,E1 -27734.931,E2 -27734.931} C_VEL
LIN {X 0,Y 184.888,Z 310.447,A -85,B 0,C 180,E1 -27735.058,E2 -27735.058} C_VEL
LIN {X 0,Y 178.461,Z 369.468,A -85,B 0,C 180,E1 -27736.423,E2 -27736.423} C_VEL
LIN {X 0,Y 175.804,Z 384.262,A -85,B 0,C 180,E1 -27736.888,E2 -27736.888} C_VEL
LIN {X 0,Y 171.762,Z 399.228,A -85,B 0,C 180,E1 -27737.481,E2 -27737.481} C_VEL
LIN {X 0,Y 166.533,Z 413.739,A -85,B 0,C 180,E1 -27738.29,E2 -27738.29} C_VEL
LIN {X 0,Y 160.14,Z 427.774,A -85,B 0,C 180,E1 -27739.353,E2 -27739.353} C_VEL
LIN {X 0,Y 153.034,Z 440.625,A -85,B 0,C 180,E1 -27740.668,E2 -27740.668} C_VEL
LIN {X 0,Y 144.464,Z 453.576,A -85,B 0,C 180,E1 -27742.444,E2 -27742.444} C_VEL
LIN {X 0,Y 136.498,Z 464.182,A -85,B 0,C 180,E1 -27744.574,E2 -27744.574} C_VEL
LIN {X 0,Y 128.165,Z 473.765,A -85,B 0,C 180,E1 -27747.001,E2 -27747.001} C_VEL
LIN {X 0,Y 118.288,Z 483.741,A -85,B 0,C 180,E1 -27750.523,E2 -27750.523} C_VEL
LIN {X 0,Y 109.089,Z 492.07,A -85,B 0,C 180,E1 -27754.783,E2 -27754.783} C_VEL
LIN {X 0,Y 100.593,Z 498.985,A -85,B 0,C 180,E1 -27759.787,E2 -27759.787} C_VEL
LIN {X 0,Y 92.142,Z 505.445,A -85,B 0,C 180,E1 -27766.658,E2 -27766.658} C_VEL
LIN {X 0,Y 85.276,Z 510.478,A -85,B 0,C 180,E1 -27774.775,E2 -27774.775} C_VEL
LIN {X 0,Y 80.374,Z 514.212,A -85,B 0,C 180,E1 -27784.082,E2 -27784.082} C_VEL
LIN {X 0,Y 77.722,Z 516.732,A -85,B 0,C 180,E1 -27794.267,E2 -27794.267} C_VEL
LIN {X 0,Y 77.567,Z 518.111,A -85,B 0,C 180,E1 -27805.306,E2 -27805.306} C_VEL
LIN {X 0,Y 77.973,Z 518.3,A -85,B 0,C 180,E1 -27810.007,E2 -27810.007} C_VEL
LIN {X 0,Y 77.584,Z 518.087,A -85,B 0,C 180,E1 -27815.204,E2 -27815.204} C_VEL
LIN {X 0,Y 77.741,Z 516.705,A -85,B 0,C 180,E1 -27825.743,E2 -27825.743} C_VEL
LIN {X 0,Y 78.456,Z 515.808,A -85,B 0,C 180,E1 -27829.87,E2 -27829.87} C_VEL
LIN {X 0,Y 78.949,Z 514.772,A -85,B 0,C 180,E1 -27834.094,E2 -27834.094} C_VEL
LIN {X 0,Y 78.92,Z 512.593,A -85,B 0,C 180,E1 -27841.13,E2 -27841.13} C_VEL
LIN {X 0,Y 79.599,Z 510.469,A -85,B 0,C 180,E1 -27846.654,E2 -27846.654} C_VEL
LIN {X 0,Y 81.311,Z 508.663,A -85,B 0,C 180,E1 -27850.478,E2 -27850.478} C_VEL
LIN {X 0,Y 82.196,Z 508.007,A -85,B 0,C 180,E1 -27851.629,E2 -27851.629} C_VEL
LIN {X 0,Y 89.229,Z 503.262,A -85,B 0,C 180,E1 -27858.447,E2 -27858.447} C_VEL
LIN {X 0,Y 98.018,Z 496.846,A -85,B 0,C 180,E1 -27864.67,E2 -27864.67} C_VEL
LIN {X 0,Y 99.934,Z 495.422,A -85,B 0,C 180,E1 -27865.764,E2 -27865.764} C_VEL
LIN {X 0,Y 91.176,Z 492.818,A -85,B 0,C 180,E1 -27877.331,E2 -27877.331} C_VEL
LIN {X 0,Y 87.86,Z 488.536,A -85,B 0,C 180,E1 -27895.412,E2 -27895.412} C_VEL
LIN {X 0,Y 92.615,Z 484.393,A -85,B 0,C 180,E1 -27909.398,E2 -27909.398} C_VEL
LIN {X 0,Y 102.253,Z 479.897,A -85,B 0,C 180,E1 -27920.544,E2 -27920.544} C_VEL
LIN {X 0,Y 115.269,Z 474.836,A -85,B 0,C 180,E1 -27929.194,E2 -27929.194} C_VEL
LIN {X 0,Y 117.984,Z 473.795,A -85,B 0,C 180,E1 -27930.468,E2 -27930.468} C_VEL
LIN {X 0,Y 116.965,Z 475,A -85,B 0,C 180,E1 -27931.407,E2 -27931.407} C_VEL
LIN {X 0,Y 107.913,Z 482.623,A -85,B 0,C 180,E1 -27935.496,E2 -27935.496} C_VEL
LIN {X 0,Y 100.531,Z 488.209,A -85,B 0,C 180,E1 -27939.729,E2 -27939.729} C_VEL
LIN {X 0,Y 91.441,Z 494.324,A -85,B 0,C 180,E1 -27946.226,E2 -27946.226} C_VEL
LIN {X 0,Y 83.797,Z 499.019,A -85,B 0,C 180,E1 -27954.042,E2 -27954.042} C_VEL
LIN {X 0,Y 77.703,Z 502.449,A -85,B 0,C 180,E1 -27963.106,E2 -27963.106} C_VEL
LIN {X 0,Y 73.573,Z 504.691,A -85,B 0,C 180,E1 -27973.34,E2 -27973.34} C_VEL
LIN {X 0,Y 71.404,Z 505.827,A -85,B 0,C 180,E1 -27984.344,E2 -27984.344} C_VEL
LIN {X 0,Y 71.399,Z 505.836,A -85,B 0,C 180,E1 -27995.642,E2 -27995.642} C_VEL
LIN {X 0,Y 73.565,Z 504.732,A -85,B 0,C 180,E1 -28006.647,E2 -28006.647} C_VEL
LIN {X 0,Y 77.683,Z 502.528,A -85,B 0,C 180,E1 -28016.887,E2 -28016.887} C_VEL
LIN {X 0,Y 83.733,Z 499.147,A -85,B 0,C 180,E1 -28025.974,E2 -28025.974} C_VEL
LIN {X 0,Y 91.374,Z 494.495,A -85,B 0,C 180,E1 -28033.799,E2 -28033.799} C_VEL
LIN {X 0,Y 100.459,Z 488.416,A -85,B 0,C 180,E1 -28040.305,E2 -28040.305} C_VEL
LIN {X 0,Y 109.143,Z 481.847,A -85,B 0,C 180,E1 -28045.176,E2 -28045.176} C_VEL
LIN {X 0,Y 118.509,Z 473.862,A -85,B 0,C 180,E1 -28049.296,E2 -28049.296} C_VEL
LIN {X 0,Y 126.893,Z 465.683,A -85,B 0,C 180,E1 -28052.385,E2 -28052.385} C_VEL
LIN {X 0,Y 135.741,Z 455.796,A -85,B 0,C 180,E1 -28055.253,E2 -28055.253} C_VEL
LIN {X 0,Y 144.446,Z 444.64,A -85,B 0,C 180,E1 -28057.573,E2 -28057.573} C_VEL
LIN {X 0,Y 152.804,Z 431.979,A -85,B 0,C 180,E1 -28059.562,E2 -28059.562} C_VEL
LIN {X 0,Y 159.748,Z 419.396,A -85,B 0,C 180,E1 -28061.052,E2 -28061.052} C_VEL
LIN {X 0,Y 165.797,Z 405.93,A -85,B 0,C 180,E1 -28062.353,E2 -28062.353} C_VEL
LIN {X 0,Y 170.889,Z 391.495,A -85,B 0,C 180,E1 -28063.47,E2 -28063.47} C_VEL
LIN {X 0,Y 174.979,Z 376.045,A -85,B 0,C 180,E1 -28064.289,E2 -28064.289} C_VEL
LIN {X 0,Y 177.705,Z 360.624,A -85,B 0,C 180,E1 -28064.84,E2 -28064.84} C_VEL
LIN {X 0,Y 182.909,Z 313.189,A -85,B 0,C 180,E1 -28066.004,E2 -28066.004} C_VEL
LIN {X 0,Y 181.283,Z 308.802,A -85,B 0,C 180,E1 -28069.247,E2 -28069.247} C_VEL
LIN {X 0,Y 180.048,Z 305.492,A -85,B 0,C 180,E1 -28072.712,E2 -28072.712} C_VEL
LIN {X 0,Y 179.18,Z 302.838,A -85,B 0,C 180,E1 -28077.752,E2 -28077.752} C_VEL
LIN {X 0,Y 179.106,Z 302.811,A -85,B 0,C 180,E1 -28080.211,E2 -28080.211} C_VEL
LIN {X 0,Y 179.775,Z 305.826,A -85,B 0,C 180,E1 -28085.749,E2 -28085.749} C_VEL
LIN {X 0,Y 180.808,Z 309.203,A -85,B 0,C 180,E1 -28089.085,E2 -28089.085} C_VEL
LIN {X 0,Y 182.127,Z 313.027,A -85,B 0,C 180,E1 -28092.006,E2 -28092.006} C_VEL
LIN {X 0,Y 182.666,Z 314.678,A -85,B 0,C 180,E1 -28093.024,E2 -28093.024} C_VEL
LIN {X 0,Y 176.255,Z 371.297,A -85,B 0,C 180,E1 -28094.262,E2 -28094.262} C_VEL
LIN {X 0,Y 173.253,Z 386.392,A -85,B 0,C 180,E1 -28094.724,E2 -28094.724} C_VEL
LIN {X 0,Y 168.942,Z 401.223,A -85,B 0,C 180,E1 -28095.303,E2 -28095.303} C_VEL
LIN {X 0,Y 163.622,Z 415.135,A -85,B 0,C 180,E1 -28096.054,E2 -28096.054} C_VEL
LIN {X 0,Y 157.114,Z 428.774,A -85,B 0,C 180,E1 -28097.045,E2 -28097.045} C_VEL
LIN {X 0,Y 149.86,Z 441.334,A -85,B 0,C 180,E1 -28098.269,E2 -28098.269} C_VEL
LIN {X 0,Y 141.104,Z 454.064,A -85,B 0,C 180,E1 -28099.942,E2 -28099.942} C_VEL
LIN {X 0,Y 133.11,Z 464.259,A -85,B 0,C 180,E1 -28101.923,E2 -28101.923} C_VEL
LIN {X 0,Y 123.587,Z 474.68,A -85,B 0,C 180,E1 -28104.524,E2 -28104.524} C_VEL
LIN {X 0,Y 114.8,Z 483.151,A -85,B 0,C 180,E1 -28107.427,E2 -28107.427} C_VEL
LIN {X 0,Y 105.155,Z 491.48,A -85,B 0,C 180,E1 -28111.565,E2 -28111.565} C_VEL
LIN {X 0,Y 96.145,Z 498.393,A -85,B 0,C 180,E1 -28116.488,E2 -28116.488} C_VEL
LIN {X 0,Y 87.042,Z 504.851,A -85,B 0,C 180,E1 -28123.4,E2 -28123.4} C_VEL
LIN {X 0,Y 79.482,Z 509.882,A -85,B 0,C 180,E1 -28131.769,E2 -28131.769} C_VEL
LIN {X 0,Y 73.951,Z 513.617,A -85,B 0,C 180,E1 -28141.637,E2 -28141.637} C_VEL
LIN {X 0,Y 70.81,Z 516.137,A -85,B 0,C 180,E1 -28152.685,E2 -28152.685} C_VEL
LIN {X 0,Y 70.491,Z 517.55,A -85,B 0,C 180,E1 -28165.553,E2 -28165.553} C_VEL
LIN {X 0,Y 70.881,Z 517.714,A -85,B 0,C 180,E1 -28170.007,E2 -28170.007} C_VEL
LIN {X 0,Y 70.435,Z 517.493,A -85,B 0,C 180,E1 -28175.734,E2 -28175.734} C_VEL
LIN {X 0,Y 70.827,Z 516.108,A -85,B 0,C 180,E1 -28187.326,E2 -28187.326} C_VEL
LIN {X 0,Y 73.948,Z 513.559,A -85,B 0,C 180,E1 -28198.38,E2 -28198.38} C_VEL
LIN {X 0,Y 79.488,Z 509.789,A -85,B 0,C 180,E1 -28208.244,E2 -28208.244} C_VEL
LIN {X 0,Y 82.196,Z 508.007,A -85,B 0,C 180,E1 -28211.629,E2 -28211.629} C_VEL
LIN {X 0,Y 83.615,Z 506.688,A -85,B 0,C 180,E1 -28214.03,E2 -28214.03} C_VEL
LIN {X 0,Y 84.628,Z 504.474,A -85,B 0,C 180,E1 -28218.317,E2 -28218.317} C_VEL
LIN {X 0,Y 86.022,Z 502.113,A -85,B 0,C 180,E1 -28222.459,E2 -28222.459} C_VEL
LIN {X 0,Y 87.937,Z 500.462,A -85,B 0,C 180,E1 -28224.504,E2 -28224.504} C_VEL
LIN {X 0,Y 89.25,Z 499.582,A -85,B 0,C 180,E1 -28225.394,E2 -28225.394} C_VEL
LIN {X 0,Y 91.064,Z 497.931,A -85,B 0,C 180,E1 -28227.301,E2 -28227.301} C_VEL
LIN {X 0,Y 83.425,Z 495.212,A -85,B 0,C 180,E1 -28240.308,E2 -28240.308} C_VEL
LIN {X 0,Y 82.369,Z 490.918,A -85,B 0,C 180,E1 -28260.001,E2 -28260.001} C_VEL
LIN {X 0,Y 88.779,Z 486.977,A -85,B 0,C 180,E1 -28273.739,E2 -28273.739} C_VEL
LIN {X 0,Y 104.855,Z 480.809,A -85,B 0,C 180,E1 -28287.982,E2 -28287.982} C_VEL
LIN {X 0,Y 107.962,Z 479.747,A -85,B 0,C 180,E1 -28289.782,E2 -28289.782} C_VEL
LIN {X 0,Y 106.701,Z 481.093,A -85,B 0,C 180,E1 -28291.092,E2 -28291.092} C_VEL
LIN {X 0,Y 98.949,Z 486.863,A -85,B 0,C 180,E1 -28294.85,E2 -28294.85} C_VEL
LIN {X 0,Y 88.828,Z 493.529,A -85,B 0,C 180,E1 -28301.26,E2 -28301.26} C_VEL
LIN {X 0,Y 80.093,Z 498.585,A -85,B 0,C 180,E1 -28308.836,E2 -28308.836} C_VEL
LIN {X 0,Y 74.575,Z 501.474,A -85,B 0,C 180,E1 -28315.559,E2 -28315.559} C_VEL
LIN {X 0,Y 68.824,Z 504.302,A -85,B 0,C 180,E1 -28325.884,E2 -28325.884} C_VEL
LIN {X 0,Y 65.326,Z 505.978,A -85,B 0,C 180,E1 -28337.567,E2 -28337.567} C_VEL
LIN {X 0,Y 64.08,Z 506.559,A -85,B 0,C 180,E1 -28349.992,E2 -28349.992} C_VEL
LIN {X 0,Y 65.318,Z 506.003,A -85,B 0,C 180,E1 -28362.419,E2 -28362.419} C_VEL
LIN {X 0,Y 68.815,Z 504.36,A -85,B 0,C 180,E1 -28374.103,E2 -28374.103} C_VEL
LIN {X 0,Y 74.524,Z 501.576,A -85,B 0,C 180,E1 -28384.451,E2 -28384.451} C_VEL
LIN {X 0,Y 82.087,Z 497.57,A -85,B 0,C 180,E1 -28393.221,E2 -28393.221} C_VEL
LIN {X 0,Y 91.152,Z 492.219,A -85,B 0,C 180,E1 -28400.436,E2 -28400.436} C_VEL
LIN {X 0,Y 101.215,Z 485.39,A -85,B 0,C 180,E1 -28406.422,E2 -28406.422} C_VEL
LIN {X 0,Y 110.816,Z 478.033,A -85,B 0,C 180,E1 -28410.685,E2 -28410.685} C_VEL
LIN {X 0,Y 120.874,Z 469.147,A -85,B 0,C 180,E1 -28414.308,E2 -28414.308} C_VEL
LIN {X 0,Y 129.692,Z 460.077,A -85,B 0,C 180,E1 -28417.095,E2 -28417.095} C_VEL
LIN {X 0,Y 138.778,Z 449.304,A -85,B 0,C 180,E1 -28419.521,E2 -28419.521} C_VEL
LIN {X 0,Y 147.365,Z 437.466,A -85,B 0,C 180,E1 -28421.404,E2 -28421.404} C_VEL
LIN {X 0,Y 154.412,Z 425.866,A -85,B 0,C 180,E1 -28422.889,E2 -28422.889} C_VEL
LIN {X 0,Y 161.342,Z 412.188,A -85,B 0,C 180,E1 -28424.221,E2 -28424.221} C_VEL
LIN {X 0,Y 167.044,Z 397.95,A -85,B 0,C 180,E1 -28425.378,E2 -28425.378} C_VEL
LIN {X 0,Y 171.41,Z 383.864,A -85,B 0,C 180,E1 -28426.204,E2 -28426.204} C_VEL
LIN {X 0,Y 174.847,Z 368.371,A -85,B 0,C 180,E1 -28426.849,E2 -28426.849} C_VEL
LIN {X 0,Y 177.276,Z 350.209,A -85,B 0,C 180,E1 -28427.352,E2 -28427.352} C_VEL
LIN {X 0,Y 180.854,Z 317.787,A -85,B 0,C 180,E1 -28428.103,E2 -28428.103} C_VEL
LIN {X 0,Y 179.585,Z 314.044,A -85,B 0,C 180,E1 -28431.277,E2 -28431.277} C_VEL
LIN {X 0,Y 178.899,Z 312.121,A -85,B 0,C 180,E1 -28433.656,E2 -28433.656} C_VEL
LIN {X 0,Y 178.311,Z 309.926,A -85,B 0,C 180,E1 -28437.741,E2 -28437.741} C_VEL
LIN {X 0,Y 178.226,Z 310.052,A -85,B 0,C 180,E1 -28440.423,E2 -28440.423} C_VEL
LIN {X 0,Y 178.773,Z 312.718,A -85,B 0,C 180,E1 -28445.286,E2 -28445.286} C_VEL
LIN {X 0,Y 179.641,Z 315.917,A -85,B 0,C 180,E1 -28448.436,E2 -28448.436} C_VEL
LIN {X 0,Y 180.657,Z 319.173,A -85,B 0,C 180,E1 -28450.961,E2 -28450.961} C_VEL
LIN {X 0,Y 174.553,Z 371.409,A -85,B 0,C 180,E1 -28452.015,E2 -28452.015} C_VEL
LIN {X 0,Y 171.377,Z 386.746,A -85,B 0,C 180,E1 -28452.455,E2 -28452.455} C_VEL
LIN {X 0,Y 166.792,Z 401.936,A -85,B 0,C 180,E1 -28453.007,E2 -28453.007} C_VEL
LIN {X 0,Y 160.969,Z 416.514,A -85,B 0,C 180,E1 -28453.74,E2 -28453.74} C_VEL
LIN {X 0,Y 154.352,Z 429.771,A -85,B 0,C 180,E1 -28454.649,E2 -28454.649} C_VEL
LIN {X 0,Y 146.154,Z 443.323,A -85,B 0,C 180,E1 -28455.918,E2 -28455.918} C_VEL
LIN {X 0,Y 137.232,Z 455.615,A -85,B 0,C 180,E1 -28457.492,E2 -28457.492} C_VEL
LIN {X 0,Y 128.161,Z 466.476,A -85,B 0,C 180,E1 -28459.602,E2 -28459.602} C_VEL
LIN {X 0,Y 117.705,Z 477.078,A -85,B 0,C 180,E1 -28462.272,E2 -28462.272} C_VEL
LIN {X 0,Y 107.282,Z 486.302,A -85,B 0,C 180,E1 -28465.754,E2 -28465.754} C_VEL
LIN {X 0,Y 97.415,Z 493.995,A -85,B 0,C 180,E1 -28470.044,E2 -28470.044} C_VEL
LIN {X 0,Y 89.475,Z 499.559,A -85,B 0,C 180,E1 -28474.448,E2 -28474.448} C_VEL
LIN {X 0,Y 80.021,Z 505.654,A -85,B 0,C 180,E1 -28481.719,E2 -28481.719} C_VEL
LIN {X 0,Y 73.944,Z 509.286,A -85,B 0,C 180,E1 -28488.304,E2 -28488.304} C_VEL
LIN {X 0,Y 67.689,Z 513.021,A -85,B 0,C 180,E1 -28498.735,E2 -28498.735} C_VEL
LIN {X 0,Y 63.975,Z 515.542,A -85,B 0,C 180,E1 -28510.766,E2 -28510.766} C_VEL
LIN {X 0,Y 63.251,Z 516.902,A -85,B 0,C 180,E1 -28523.629,E2 -28523.629} C_VEL
LIN {X 0,Y 63.787,Z 517.128,A -85,B 0,C 180,E1 -28530.008,E2 -28530.008} C_VEL
LIN {X 0,Y 63.303,Z 516.9,A -85,B 0,C 180,E1 -28536.382,E2 -28536.382} C_VEL
LIN {X 0,Y 63.991,Z 515.513,A -85,B 0,C 180,E1 -28549.246,E2 -28549.246} C_VEL
LIN {X 0,Y 67.683,Z 512.962,A -85,B 0,C 180,E1 -28561.286,E2 -28561.286} C_VEL
LIN {X 0,Y 73.955,Z 509.193,A -85,B 0,C 180,E1 -28571.708,E2 -28571.708} C_VEL
LIN {X 0,Y 82.275,Z 504.131,A -85,B 0,C 180,E1 -28580.254,E2 -28580.254} C_VEL
LIN {X 0,Y 87.937,Z 500.462,A -85,B 0,C 180,E1 -28584.504,E2 -28584.504} C_VEL
LIN {X 0,Y 88.496,Z 499.742,A -85,B 0,C 180,E1 -28585.569,E2 -28585.569} C_VEL
LIN {X 0,Y 87.988,Z 499.13,A -85,B 0,C 180,E1 -28587.149,E2 -28587.149} C_VEL
LIN {X 0,Y 86.062,Z 498.761,A -85,B 0,C 180,E1 -28589.34,E2 -28589.34} C_VEL
LIN {X 0,Y 78.948,Z 498.81,A -85,B 0,C 180,E1 -28595.574,E2 -28595.574} C_VEL
LIN {X 0,Y 77.861,Z 498.565,A -85,B 0,C 180,E1 -28597.457,E2 -28597.457} C_VEL
LIN {X 0,Y 75.168,Z 495.346,A -85,B 0,C 180,E1 -28614.636,E2 -28614.636} C_VEL
LIN {X 0,Y 79.669,Z 491.793,A -85,B 0,C 180,E1 -28630.162,E2 -28630.162} C_VEL
LIN {X 0,Y 93.948,Z 486.378,A -85,B 0,C 180,E1 -28646.133,E2 -28646.133} C_VEL
LIN {X 0,Y 98.153,Z 485.014,A -85,B 0,C 180,E1 -28649.009,E2 -28649.009} C_VEL
LIN {X 0,Y 97.545,Z 485.748,A -85,B 0,C 180,E1 -28650.155,E2 -28650.155} C_VEL
LIN {X 0,Y 86.88,Z 492.617,A -85,B 0,C 180,E1 -28655.999,E2 -28655.999} C_VEL
LIN {X 0,Y 77.131,Z 498.008,A -85,B 0,C 180,E1 -28663.193,E2 -28663.193} C_VEL
LIN {X 0,Y 68.851,Z 502.059,A -85,B 0,C 180,E1 -28672.224,E2 -28672.224} C_VEL
LIN {X 0,Y 62.441,Z 504.887,A -85,B 0,C 180,E1 -28683.233,E2 -28683.233} C_VEL
LIN {X 0,Y 58.451,Z 506.562,A -85,B 0,C 180,E1 -28696.077,E2 -28696.077} C_VEL
LIN {X 0,Y 57.018,Z 507.143,A -85,B 0,C 180,E1 -28709.991,E2 -28709.991} C_VEL
LIN {X 0,Y 58.444,Z 506.586,A -85,B 0,C 180,E1 -28723.907,E2 -28723.907} C_VEL
LIN {X 0,Y 62.43,Z 504.944,A -85,B 0,C 180,E1 -28736.753,E2 -28736.753} C_VEL
LIN {X 0,Y 68.805,Z 502.16,A -85,B 0,C 180,E1 -28747.787,E2 -28747.787} C_VEL
LIN {X 0,Y 77.076,Z 498.154,A -85,B 0,C 180,E1 -28756.831,E2 -28756.831} C_VEL
LIN {X 0,Y 86.815,Z 492.802,A -85,B 0,C 180,E1 -28764.04,E2 -28764.04} C_VEL
LIN {X 0,Y 97.472,Z 485.972,A -85,B 0,C 180,E1 -28769.898,E2 -28769.898} C_VEL
LIN {X 0,Y 107.526,Z 478.613,A -85,B 0,C 180,E1 -28773.977,E2 -28773.977} C_VEL
LIN {X 0,Y 117.969,Z 469.728,A -85,B 0,C 180,E1 -28777.417,E2 -28777.417} C_VEL
LIN {X 0,Y 127.104,Z 460.654,A -85,B 0,C 180,E1 -28780.036,E2 -28780.036} C_VEL
LIN {X 0,Y 134.881,Z 451.782,A -85,B 0,C 180,E1 -28781.961,E2 -28781.961} C_VEL
LIN {X 0,Y 143.659,Z 440.329,A -85,B 0,C 180,E1 -28783.742,E2 -28783.742} C_VEL
LIN {X 0,Y 151.67,Z 427.825,A -85,B 0,C 180,E1 -28785.291,E2 -28785.291} C_VEL
LIN {X 0,Y 158.155,Z 415.747,A -85,B 0,C 180,E1 -28786.41,E2 -28786.41} C_VEL
LIN {X 0,Y 163.926,Z 402.488,A -85,B 0,C 180,E1 -28787.483,E2 -28787.483} C_VEL
LIN {X 0,Y 168.64,Z 388.784,A -85,B 0,C 180,E1 -28788.318,E2 -28788.318} C_VEL
LIN {X 0,Y 172.485,Z 373.624,A -85,B 0,C 180,E1 -28788.966,E2 -28788.966} C_VEL
LIN {X 0,Y 175.054,Z 357.847,A -85,B 0,C 180,E1 -28789.419,E2 -28789.419} C_VEL
LIN {X 0,Y 179.041,Z 322.621,A -85,B 0,C 180,E1 -28790.202,E2 -28790.202} C_VEL
LIN {X 0,Y 178.083,Z 319.369,A -85,B 0,C 180,E1 -28793.414,E2 -28793.414} C_VEL
LIN {X 0,Y 177.443,Z 317.002,A -85,B 0,C 180,E1 -28797.73,E2 -28797.73} C_VEL
LIN {X 0,Y 177.349,Z 317.191,A -85,B 0,C 180,E1 -28800.425,E2 -28800.425} C_VEL
LIN {X 0,Y 177.784,Z 319.596,A -85,B 0,C 180,E1 -28804.818,E2 -28804.818} C_VEL
LIN {X 0,Y 178.546,Z 322.763,A -85,B 0,C 180,E1 -28807.918,E2 -28807.918} C_VEL
LIN {X 0,Y 178.844,Z 323.747,A -85,B 0,C 180,E1 -28808.788,E2 -28808.788} C_VEL
LIN {X 0,Y 173.246,Z 370.688,A -85,B 0,C 180,E1 -28809.709,E2 -28809.709} C_VEL
LIN {X 0,Y 169.984,Z 386.213,A -85,B 0,C 180,E1 -28810.112,E2 -28810.112} C_VEL
LIN {X 0,Y 165.337,Z 401.385,A -85,B 0,C 180,E1 -28810.608,E2 -28810.608} C_VEL
LIN {X 0,Y 159.433,Z 415.952,A -85,B 0,C 180,E1 -28811.262,E2 -28811.262} C_VEL
LIN {X 0,Y 152.711,Z 429.203,A -85,B 0,C 180,E1 -28812.071,E2 -28812.071} C_VEL
LIN {X 0,Y 144.364,Z 442.749,A -85,B 0,C 180,E1 -28813.2,E2 -28813.2} C_VEL
LIN {X 0,Y 135.249,Z 455.033,A -85,B 0,C 180,E1 -28814.592,E2 -28814.592} C_VEL
LIN {X 0,Y 126.301,Z 465.488,A -85,B 0,C 180,E1 -28816.45,E2 -28816.45} C_VEL
LIN {X 0,Y 116.775,Z 475.003,A -85,B 0,C 180,E1 -28818.591,E2 -28818.591} C_VEL
LIN {X 0,Y 105.872,Z 484.466,A -85,B 0,C 180,E1 -28821.681,E2 -28821.681} C_VEL
LIN {X 0,Y 95.465,Z 492.378,A -85,B 0,C 180,E1 -28825.614,E2 -28825.614} C_VEL
LIN {X 0,Y 85.601,Z 498.966,A -85,B 0,C 180,E1 -28830.463,E2 -28830.463} C_VEL
LIN {X 0,Y 75.409,Z 505.06,A -85,B 0,C 180,E1 -28837.622,E2 -28837.622} C_VEL
LIN {X 0,Y 68.743,Z 508.693,A -85,B 0,C 180,E1 -28844.314,E2 -28844.314} C_VEL
LIN {X 0,Y 61.635,Z 512.426,A -85,B 0,C 180,E1 -28855.251,E2 -28855.251} C_VEL
LIN {X 0,Y 57.243,Z 514.949,A -85,B 0,C 180,E1 -28868.398,E2 -28868.398} C_VEL
LIN {X 0,Y 56.117,Z 516.308,A -85,B 0,C 180,E1 -28882.815,E2 -28882.815} C_VEL
LIN {X 0,Y 56.69,Z 516.541,A -85,B 0,C 180,E1 -28890.009,E2 -28890.009} C_VEL
LIN {X 0,Y 56.177,Z 516.307,A -85,B 0,C 180,E1 -28897.196,E2 -28897.196} C_VEL
LIN {X 0,Y 57.257,Z 514.919,A -85,B 0,C 180,E1 -28911.616,E2 -28911.616} C_VEL
LIN {X 0,Y 61.63,Z 512.365,A -85,B 0,C 180,E1 -28924.772,E2 -28924.772} C_VEL
LIN {X 0,Y 68.756,Z 508.598,A -85,B 0,C 180,E1 -28935.696,E2 -28935.696} C_VEL
LIN {X 0,Y 77.862,Z 503.535,A -85,B 0,C 180,E1 -28944.337,E2 -28944.337} C_VEL
LIN {X 0,Y 82.978,Z 500.482,A -85,B 0,C 180,E1 -28947.894,E2 -28947.894} C_VEL
LIN {X 0,Y 82.326,Z 500.131,A -85,B 0,C 180,E1 -28949.19,E2 -28949.19} C_VEL
LIN {X 0,Y 77.861,Z 498.565,A -85,B 0,C 180,E1 -28957.457,E2 -28957.457} C_VEL
LIN {X 0,Y 75.842,Z 498.058,A -85,B 0,C 180,E1 -28961.583,E2 -28961.583} C_VEL
LIN {X 0,Y 69.697,Z 497.76,A -85,B 0,C 180,E1 -28974.796,E2 -28974.796} C_VEL
LIN {X 0,Y 69.361,Z 497.298,A -85,B 0,C 180,E1 -28979.619,E2 -28979.619} C_VEL
LIN {X 0,Y 69.613,Z 497.031,A -85,B 0,C 180,E1 -28981.207,E2 -28981.207} C_VEL
LIN {X 0,Y 76.21,Z 493.754,A -85,B 0,C 180,E1 -28996.061,E2 -28996.061} C_VEL
LIN {X 0,Y 88.649,Z 489.696,A -85,B 0,C 180,E1 -29008.404,E2 -29008.404} C_VEL
LIN {X 0,Y 88.446,Z 489.969,A -85,B 0,C 180,E1 -29009.054,E2 -29009.054} C_VEL
LIN {X 0,Y 80.187,Z 494.701,A -85,B 0,C 180,E1 -29013.62,E2 -29013.62} C_VEL
LIN {X 0,Y 70.06,Z 499.755,A -85,B 0,C 180,E1 -29021.195,E2 -29021.195} C_VEL
LIN {X 0,Y 63.406,Z 502.644,A -85,B 0,C 180,E1 -29028.304,E2 -29028.304} C_VEL
LIN {X 0,Y 56.214,Z 505.471,A -85,B 0,C 180,E1 -29039.984,E2 -29039.984} C_VEL
LIN {X 0,Y 51.627,Z 507.145,A -85,B 0,C 180,E1 -29054.191,E2 -29054.191} C_VEL
LIN {X 0,Y 49.958,Z 507.727,A -85,B 0,C 180,E1 -29069.99,E2 -29069.99} C_VEL
LIN {X 0,Y 51.62,Z 507.169,A -85,B 0,C 180,E1 -29085.791,E2 -29085.791} C_VEL
LIN {X 0,Y 56.201,Z 505.528,A -85,B 0,C 180,E1 -29100.003,E2 -29100.003} C_VEL
LIN {X 0,Y 63.343,Z 502.745,A -85,B 0,C 180,E1 -29111.725,E2 -29111.725} C_VEL
LIN {X 0,Y 72.398,Z 498.74,A -85,B 0,C 180,E1 -29120.938,E2 -29120.938} C_VEL
LIN {X 0,Y 82.856,Z 493.384,A -85,B 0,C 180,E1 -29128.006,E2 -29128.006} C_VEL
LIN {X 0,Y 94.113,Z 486.556,A -85,B 0,C 180,E1 -29133.639,E2 -29133.639} C_VEL
LIN {X 0,Y 104.614,Z 479.194,A -85,B 0,C 180,E1 -29137.464,E2 -29137.464} C_VEL
LIN {X 0,Y 115.432,Z 470.307,A -85,B 0,C 180,E1 -29140.669,E2 -29140.669} C_VEL
LIN {X 0,Y 125.87,Z 460.188,A -85,B 0,C 180,E1 -29143.325,E2 -29143.325} C_VEL
LIN {X 0,Y 135.305,Z 449.485,A -85,B 0,C 180,E1 -29145.317,E2 -29145.317} C_VEL
LIN {X 0,Y 144.303,Z 437.451,A -85,B 0,C 180,E1 -29146.903,E2 -29146.903} C_VEL
LIN {X 0,Y 151.688,Z 425.607,A -85,B 0,C 180,E1 -29148.152,E2 -29148.152} C_VEL
LIN {X 0,Y 158.633,Z 412.168,A -85,B 0,C 180,E1 -29149.245,E2 -29149.245} C_VEL
LIN {X 0,Y 164.458,Z 397.963,A -85,B 0,C 180,E1 -29150.23,E2 -29150.23} C_VEL
LIN {X 0,Y 169.014,Z 383.473,A -85,B 0,C 180,E1 -29150.937,E2 -29150.937} C_VEL
LIN {X 0,Y 172.35,Z 368.523,A -85,B 0,C 180,E1 -29151.458,E2 -29151.458} C_VEL
LIN {X 0,Y 175.028,Z 348.526,A -85,B 0,C 180,E1 -29151.928,E2 -29151.928} C_VEL
LIN {X 0,Y 177.433,Z 327.659,A -85,B 0,C 180,E1 -29152.377,E2 -29152.377} C_VEL
LIN {X 0,Y 176.928,Z 325.869,A -85,B 0,C 180,E1 -29154.586,E2 -29154.586} C_VEL
LIN {X 0,Y 176.567,Z 324.139,A -85,B 0,C 180,E1 -29157.719,E2 -29157.719} C_VEL
LIN {X 0,Y 176.477,Z 324.292,A -85,B 0,C 180,E1 -29160.428,E2 -29160.428} C_VEL
LIN {X 0,Y 176.815,Z 326.565,A -85,B 0,C 180,E1 -29164.417,E2 -29164.417} C_VEL
LIN {X 0,Y 177.261,Z 328.783,A -85,B 0,C 180,E1 -29166.639,E2 -29166.639} C_VEL
LIN {X 0,Y 172.189,Z 370.197,A -85,B 0,C 180,E1 -29167.375,E2 -29167.375} C_VEL
LIN {X 0,Y 168.883,Z 385.682,A -85,B 0,C 180,E1 -29167.742,E2 -29167.742} C_VEL
LIN {X 0,Y 164.177,Z 400.832,A -85,B 0,C 180,E1 -29168.168,E2 -29168.168} C_VEL
LIN {X 0,Y 158.199,Z 415.39,A -85,B 0,C 180,E1 -29168.74,E2 -29168.74} C_VEL
LIN {X 0,Y 151.382,Z 428.634,A -85,B 0,C 180,E1 -29169.435,E2 -29169.435} C_VEL
LIN {X 0,Y 142.903,Z 442.173,A -85,B 0,C 180,E1 -29170.412,E2 -29170.412} C_VEL
LIN {X 0,Y 133.637,Z 454.457,A -85,B 0,C 180,E1 -29171.645,E2 -29171.645} C_VEL
LIN {X 0,Y 124.033,Z 465.364,A -85,B 0,C 180,E1 -29173.358,E2 -29173.358} C_VEL
LIN {X 0,Y 113.064,Z 475.91,A -85,B 0,C 180,E1 -29175.554,E2 -29175.554} C_VEL
LIN {X 0,Y 101.858,Z 485.122,A -85,B 0,C 180,E1 -29178.445,E2 -29178.445} C_VEL
LIN {X 0,Y 91.07,Z 492.813,A -85,B 0,C 180,E1 -29182.188,E2 -29182.188} C_VEL
LIN {X 0,Y 79.344,Z 500.029,A -85,B 0,C 180,E1 -29187.669,E2 -29187.669} C_VEL
LIN {X 0,Y 68.698,Z 505.753,A -85,B 0,C 180,E1 -29195.086,E2 -29195.086} C_VEL
LIN {X 0,Y 59.492,Z 510.172,A -85,B 0,C 180,E1 -29205.136,E2 -29205.136} C_VEL
LIN {X 0,Y 52.841,Z 513.241,A -85,B 0,C 180,E1 -29217.871,E2 -29217.871} C_VEL
LIN {X 0,Y 49.341,Z 515.18,A -85,B 0,C 180,E1 -29233.46,E2 -29233.46} C_VEL
LIN {X 0,Y 49.567,Z 515.952,A -85,B 0,C 180,E1 -29250.01,E2 -29250.01} C_VEL
LIN {X 0,Y 49.078,Z 515.715,A -85,B 0,C 180,E1 -29258.244,E2 -29258.244} C_VEL
LIN {X 0,Y 50.638,Z 514.325,A -85,B 0,C 180,E1 -29274.616,E2 -29274.616} C_VEL
LIN {X 0,Y 55.863,Z 511.769,A -85,B 0,C 180,E1 -29288.99,E2 -29288.99} C_VEL
LIN {X 0,Y 63.933,Z 508.003,A -85,B 0,C 180,E1 -29300.32,E2 -29300.32} C_VEL
LIN {X 0,Y 73.897,Z 502.939,A -85,B 0,C 180,E1 -29308.877,E2 -29308.877} C_VEL
LIN {X 0,Y 73.695,Z 502.077,A -85,B 0,C 180,E1 -29311.522,E2 -29311.522} C_VEL
LIN {X 0,Y 68.631,Z 498.335,A -85,B 0,C 180,E1 -29334.123,E2 -29334.123} C_VEL
LIN {X 0,Y 69.613,Z 497.031,A -85,B 0,C 180,E1 -29341.207,E2 -29341.207} C_VEL
LIN {X 0,Y 70.365,Z 496.371,A -85,B 0,C 180,E1 -29345.977,E2 -29345.977} C_VEL
LIN {X 0,Y 72.919,Z 495.591,A -85,B 0,C 180,E1 -29360.109,E2 -29360.109} C_VEL
LIN {X 0,Y 75.397,Z 494.973,A -85,B 0,C 180,E1 -29364.201,E2 -29364.201} C_VEL
LIN {X 0,Y 76.514,Z 494.654,A -85,B 0,C 180,E1 -29365.392,E2 -29365.392} C_VEL
LIN {X 0,Y 78.015,Z 494.222,A -85,B 0,C 180,E1 -29366.772,E2 -29366.772} C_VEL
LIN {X 0,Y 78.189,Z 494.432,A -85,B 0,C 180,E1 -29368.307,E2 -29368.307} C_VEL
LIN {X 0,Y 68.206,Z 499.182,A -85,B 0,C 180,E1 -29374.467,E2 -29374.467} C_VEL
LIN {X 0,Y 58.297,Z 503.231,A -85,B 0,C 180,E1 -29383.658,E2 -29383.658} C_VEL
LIN {X 0,Y 50.197,Z 506.058,A -85,B 0,C 180,E1 -29395.93,E2 -29395.93} C_VEL
LIN {X 0,Y 44.876,Z 507.729,A -85,B 0,C 180,E1 -29411.735,E2 -29411.735} C_VEL
LIN {X 0,Y 42.9,Z 508.31,A -85,B 0,C 180,E1 -29429.988,E2 -29429.988} C_VEL
LIN {X 0,Y 44.868,Z 507.752,A -85,B 0,C 180,E1 -29448.245,E2 -29448.245} C_VEL
LIN {X 0,Y 50.181,Z 506.114,A -85,B 0,C 180,E1 -29464.058,E2 -29464.058} C_VEL
LIN {X 0,Y 58.244,Z 503.33,A -85,B 0,C 180,E1 -29476.372,E2 -29476.372} C_VEL
LIN {X 0,Y 68.149,Z 499.325,A -85,B 0,C 180,E1 -29485.576,E2 -29485.576} C_VEL
LIN {X 0,Y 79.33,Z 493.967,A -85,B 0,C 180,E1 -29492.35,E2 -29492.35} C_VEL
LIN {X 0,Y 91.194,Z 487.136,A -85,B 0,C 180,E1 -29497.622,E2 -29497.622} C_VEL
LIN {X 0,Y 102.111,Z 479.773,A -85,B 0,C 180,E1 -29501.133,E2 -29501.133} C_VEL
LIN {X 0,Y 113.285,Z 470.886,A -85,B 0,C 180,E1 -29504.05,E2 -29504.05} C_VEL
LIN {X 0,Y 122.986,Z 461.811,A -85,B 0,C 180,E1 -29506.259,E2 -29506.259} C_VEL
LIN {X 0,Y 132.856,Z 451.024,A -85,B 0,C 180,E1 -29508.114,E2 -29508.114} C_VEL
LIN {X 0,Y 142.037,Z 439.177,A -85,B 0,C 180,E1 -29509.528,E2 -29509.528} C_VEL
LIN {X 0,Y 149.551,Z 427.567,A -85,B 0,C 180,E1 -29510.682,E2 -29510.682} C_VEL
LIN {X 0,Y 156.861,Z 413.971,A -85,B 0,C 180,E1 -29511.681,E2 -29511.681} C_VEL
LIN {X 0,Y 162.987,Z 399.607,A -85,B 0,C 180,E1 -29512.611,E2 -29512.611} C_VEL
LIN {X 0,Y 167.624,Z 385.478,A -85,B 0,C 180,E1 -29513.26,E2 -29513.26} C_VEL
LIN {X 0,Y 171.221,Z 370.163,A -85,B 0,C 180,E1 -29513.765,E2 -29513.765} C_VEL
LIN {X 0,Y 173.794,Z 352.18,A -85,B 0,C 180,E1 -29514.186,E2 -29514.186} C_VEL
LIN {X 0,Y 176.057,Z 333.044,A -85,B 0,C 180,E1 -29514.537,E2 -29514.537} C_VEL
LIN {X 0,Y 175.691,Z 331.277,A -85,B 0,C 180,E1 -29517.707,E2 -29517.707} C_VEL
LIN {X 0,Y 175.603,Z 331.416,A -85,B 0,C 180,E1 -29520.43,E2 -29520.43} C_VEL
LIN {X 0,Y 175.858,Z 333.507,A -85,B 0,C 180,E1 -29524.01,E2 -29524.01} C_VEL
LIN {X 0,Y 175.917,Z 333.905,A -85,B 0,C 180,E1 -29524.439,E2 -29524.439} C_VEL
LIN {X 0,Y 171.395,Z 369.874,A -85,B 0,C 180,E1 -29525.019,E2 -29525.019} C_VEL
LIN {X 0,Y 167.857,Z 385.947,A -85,B 0,C 180,E1 -29525.356,E2 -29525.356} C_VEL
LIN {X 0,Y 162.888,Z 401.412,A -85,B 0,C 180,E1 -29525.734,E2 -29525.734} C_VEL
LIN {X 0,Y 157.276,Z 414.828,A -85,B 0,C 180,E1 -29526.179,E2 -29526.179} C_VEL
LIN {X 0,Y 150.378,Z 428.064,A -85,B 0,C 180,E1 -29526.755,E2 -29526.755} C_VEL
LIN {X 0,Y 141.781,Z 441.594,A -85,B 0,C 180,E1 -29527.558,E2 -29527.558} C_VEL
LIN {X 0,Y 132.372,Z 453.873,A -85,B 0,C 180,E1 -29528.594,E2 -29528.594} C_VEL
LIN {X 0,Y 122.894,Z 464.423,A -85,B 0,C 180,E1 -29530.013,E2 -29530.013} C_VEL
LIN {X 0,Y 111.36,Z 475.325,A -85,B 0,C 180,E1 -29532.006,E2 -29532.006} C_VEL
LIN {X 0,Y 99.817,Z 484.533,A -85,B 0,C 180,E1 -29534.529,E2 -29534.529} C_VEL
LIN {X 0,Y 88.605,Z 492.223,A -85,B 0,C 180,E1 -29537.879,E2 -29537.879} C_VEL
LIN {X 0,Y 76.261,Z 499.435,A -85,B 0,C 180,E1 -29542.862,E2 -29542.862} C_VEL
LIN {X 0,Y 64.827,Z 505.16,A -85,B 0,C 180,E1 -29549.872,E2 -29549.872} C_VEL
LIN {X 0,Y 53.942,Z 509.855,A -85,B 0,C 180,E1 -29560.649,E2 -29560.649} C_VEL
LIN {X 0,Y 46.893,Z 512.646,A -85,B 0,C 180,E1 -29573.18,E2 -29573.18} C_VEL
LIN {X 0,Y 42.497,Z 514.586,A -85,B 0,C 180,E1 -29590.699,E2 -29590.699} C_VEL
LIN {X 0,Y 42.443,Z 515.364,A -85,B 0,C 180,E1 -29610.012,E2 -29610.012} C_VEL
LIN {X 0,Y 42.516,Z 514.569,A -85,B 0,C 180,E1 -29629.318,E2 -29629.318} C_VEL
LIN {X 0,Y 46.898,Z 512.599,A -85,B 0,C 180,E1 -29646.842,E2 -29646.842} C_VEL
LIN {X 0,Y 54.747,Z 509.445,A -85,B 0,C 180,E1 -29660.389,E2 -29660.389} C_VEL
LIN {X 0,Y 64.852,Z 505.044,A -85,B 0,C 180,E1 -29670.122,E2 -29670.122} C_VEL
LIN {X 0,Y 65.959,Z 504.028,A -85,B 0,C 180,E1 -29672.742,E2 -29672.742} C_VEL
LIN {X 0,Y 62.005,Z 501.028,A -85,B 0,C 180,E1 -29693.492,E2 -29693.492} C_VEL
LIN {X 0,Y 66.655,Z 497.858,A -85,B 0,C 180,E1 -29712.174,E2 -29712.174} C_VEL
LIN {X 0,Y 76.514,Z 494.654,A -85,B 0,C 180,E1 -29725.392,E2 -29725.392} C_VEL
LIN {X 0,Y 76.821,Z 494.715,A -85,B 0,C 180,E1 -29726.535,E2 -29726.535} C_VEL
LIN {X 0,Y 75.697,Z 495.47,A -85,B 0,C 180,E1 -29728.402,E2 -29728.402} C_VEL
LIN {X 0,Y 72.266,Z 497.174,A -85,B 0,C 180,E1 -29730.643,E2 -29730.643} C_VEL
LIN {X 0,Y 69.187,Z 498.475,A -85,B 0,C 180,E1 -29731.918,E2 -29731.918} C_VEL
LIN {X 0,Y 59.755,Z 501.877,A -85,B 0,C 180,E1 -29735.056,E2 -29735.056} C_VEL
LIN {X 0,Y 53.18,Z 503.996,A -85,B 0,C 180,E1 -29738.881,E2 -29738.881} C_VEL
LIN {X 0,Y 51.298,Z 504.556,A -85,B 0,C 180,E1 -29740.764,E2 -29740.764} C_VEL
LIN {X 0,Y 44.514,Z 506.643,A -85,B 0,C 180,E1 -29750.822,E2 -29750.822} C_VEL
LIN {X 0,Y 38.236,Z 508.312,A -85,B 0,C 180,E1 -29768.418,E2 -29768.418} C_VEL
LIN {X 0,Y 35.842,Z 508.893,A -85,B 0,C 180,E1 -29789.986,E2 -29789.986} C_VEL
LIN {X 0,Y 38.227,Z 508.335,A -85,B 0,C 180,E1 -29811.559,E2 -29811.559} C_VEL
LIN {X 0,Y 44.497,Z 506.698,A -85,B 0,C 180,E1 -29829.166,E2 -29829.166} C_VEL
LIN {X 0,Y 53.604,Z 503.914,A -85,B 0,C 180,E1 -29841.858,E2 -29841.858} C_VEL
LIN {X 0,Y 64.407,Z 499.909,A -85,B 0,C 180,E1 -29850.786,E2 -29850.786} C_VEL
LIN {X 0,Y 76.301,Z 494.55,A -85,B 0,C 180,E1 -29857.068,E2 -29857.068} C_VEL
LIN {X 0,Y 88.741,Z 487.718,A -85,B 0,C 180,E1 -29861.852,E2 -29861.852} C_VEL
LIN {X 0,Y 100.045,Z 480.354,A -85,B 0,C 180,E1 -29864.976,E2 -29864.976} C_VEL
LIN {X 0,Y 111.544,Z 471.466,A -85,B 0,C 180,E1 -29867.557,E2 -29867.557} C_VEL
LIN {X 0,Y 121.496,Z 462.39,A -85,B 0,C 180,E1 -29869.512,E2 -29869.512} C_VEL
LIN {X 0,Y 131.581,Z 451.599,A -85,B 0,C 180,E1 -29871.132,E2 -29871.132} C_VEL
LIN {X 0,Y 140.923,Z 439.748,A -85,B 0,C 180,E1 -29872.358,E2 -29872.358} C_VEL
LIN {X 0,Y 148.571,Z 428.134,A -85,B 0,C 180,E1 -29873.37,E2 -29873.37} C_VEL
LIN {X 0,Y 155.977,Z 414.568,A -85,B 0,C 180,E1 -29874.248,E2 -29874.248} C_VEL
LIN {X 0,Y 161.687,Z 401.547,A -85,B 0,C 180,E1 -29875.013,E2 -29875.013} C_VEL
LIN {X 0,Y 166.728,Z 386.749,A -85,B 0,C 180,E1 -29875.642,E2 -29875.642} C_VEL
LIN {X 0,Y 170.369,Z 371.824,A -85,B 0,C 180,E1 -29876.106,E2 -29876.106} C_VEL
LIN {X 0,Y 173.033,Z 354.178,A -85,B 0,C 180,E1 -29876.501,E2 -29876.501} C_VEL
LIN {X 0,Y 174.864,Z 338.959,A -85,B 0,C 180,E1 -29876.763,E2 -29876.763} C_VEL
LIN {X 0,Y 174.814,Z 338.425,A -85,B 0,C 180,E1 -29877.696,E2 -29877.696} C_VEL
LIN {X 0,Y 174.726,Z 338.507,A -85,B 0,C 180,E1 -29880.288,E2 -29880.288} C_VEL
LIN {X 0,Y 174.785,Z 339.436,A -85,B 0,C 180,E1 -29882.201,E2 -29882.201} C_VEL
LIN {X 0,Y 170.921,Z 369.379,A -85,B 0,C 180,E1 -29882.65,E2 -29882.65} C_VEL
LIN {X 0,Y 167.344,Z 385.408,A -85,B 0,C 180,E1 -29882.936,E2 -29882.936} C_VEL
LIN {X 0,Y 162.331,Z 400.856,A -85,B 0,C 180,E1 -29883.232,E2 -29883.232} C_VEL
LIN {X 0,Y 156.67,Z 414.265,A -85,B 0,C 180,E1 -29883.593,E2 -29883.593} C_VEL
LIN {X 0,Y 149.707,Z 427.494,A -85,B 0,C 180,E1 -29884.042,E2 -29884.042} C_VEL
LIN {X 0,Y 141.021,Z 441.018,A -85,B 0,C 180,E1 -29884.684,E2 -29884.684} C_VEL
LIN {X 0,Y 131.499,Z 453.297,A -85,B 0,C 180,E1 -29885.532,E2 -29885.532} C_VEL
LIN {X 0,Y 122.212,Z 463.448,A -85,B 0,C 180,E1 -29886.604,E2 -29886.604} C_VEL
LIN {X 0,Y 113.494,Z 471.751,A -85,B 0,C 180,E1 -29887.822,E2 -29887.822} C_VEL
LIN {X 0,Y 101.618,Z 481.456,A -85,B 0,C 180,E1 -29889.787,E2 -29889.787} C_VEL
LIN {X 0,Y 89.955,Z 489.582,A -85,B 0,C 180,E1 -29892.449,E2 -29892.449} C_VEL
LIN {X 0,Y 76.93,Z 497.187,A -85,B 0,C 180,E1 -29896.442,E2 -29896.442} C_VEL
LIN {X 0,Y 64.528,Z 503.279,A -85,B 0,C 180,E1 -29902.237,E2 -29902.237} C_VEL
LIN {X 0,Y 53.083,Z 507.99,A -85,B 0,C 180,E1 -29910.639,E2 -29910.639} C_VEL
LIN {X 0,Y 45.579,Z 510.643,A -85,B 0,C 180,E1 -29919.578,E2 -29919.578} C_VEL
LIN {X 0,Y 37.999,Z 513.165,A -85,B 0,C 180,E1 -29936.316,E2 -29936.316} C_VEL
LIN {X 0,Y 34.895,Z 514.532,A -85,B 0,C 180,E1 -29958.396,E2 -29958.396} C_VEL
LIN {X 0,Y 35.317,Z 514.775,A -85,B 0,C 180,E1 -29970.015,E2 -29970.015} C_VEL
LIN {X 0,Y 35.82,Z 513.975,A -85,B 0,C 180,E1 -29993.119,E2 -29993.119} C_VEL
LIN {X 0,Y 41.363,Z 512.004,A -85,B 0,C 180,E1 -30012.832,E2 -30012.832} C_VEL
LIN {X 0,Y 50.46,Z 508.85,A -85,B 0,C 180,E1 -30026.703,E2 -30026.703} C_VEL
LIN {X 0,Y 57.193,Z 506.276,A -85,B 0,C 180,E1 -30032.858,E2 -30032.858} C_VEL
LIN {X 0,Y 57.698,Z 505.572,A -85,B 0,C 180,E1 -30035.7,E2 -30035.7} C_VEL
LIN {X 0,Y 56.273,Z 502.196,A -85,B 0,C 180,E1 -30062.187,E2 -30062.187} C_VEL
LIN {X 0,Y 67.413,Z 498.257,A -85,B 0,C 180,E1 -30084.647,E2 -30084.647} C_VEL
LIN {X 0,Y 68.355,Z 498.001,A -85,B 0,C 180,E1 -30085.695,E2 -30085.695} C_VEL
LIN {X 0,Y 66.505,Z 498.914,A -85,B 0,C 180,E1 -30087.942,E2 -30087.942} C_VEL
LIN {X 0,Y 58.901,Z 501.951,A -85,B 0,C 180,E1 -30093.345,E2 -30093.345} C_VEL
LIN {X 0,Y 51.298,Z 504.556,A -85,B 0,C 180,E1 -30100.764,E2 -30100.764} C_VEL
LIN {X 0,Y 47.007,Z 505.856,A -85,B 0,C 180,E1 -30105.279,E2 -30105.279} C_VEL
LIN {X 0,Y 39.206,Z 507.631,A -85,B 0,C 180,E1 -30113.115,E2 -30113.115} C_VEL
LIN {X 0,Y 33.448,Z 508.674,A -85,B 0,C 180,E1 -30121.709,E2 -30121.709} C_VEL
LIN {X 0,Y 30.379,Z 509.156,A -85,B 0,C 180,E1 -30130.822,E2 -30130.822} C_VEL
LIN {X 0,Y 29.773,Z 509.268,A -85,B 0,C 180,E1 -30134.407,E2 -30134.407} C_VEL
LIN {X 0,Y 29.55,Z 509.335,A -85,B 0,C 180,E1 -30163.741,E2 -30163.741} C_VEL
LIN {X 0,Y 35.062,Z 508.239,A -85,B 0,C 180,E1 -30186.946,E2 -30186.946} C_VEL
LIN {X 0,Y 44.151,Z 506.039,A -85,B 0,C 180,E1 -30202.721,E2 -30202.721} C_VEL
LIN {X 0,Y 55.279,Z 502.654,A -85,B 0,C 180,E1 -30212.846,E2 -30212.846} C_VEL
LIN {X 0,Y 67.437,Z 497.998,A -85,B 0,C 180,E1 -30219.686,E2 -30219.686} C_VEL
LIN {X 0,Y 80.258,Z 491.916,A -85,B 0,C 180,E1 -30224.392,E2 -30224.392} C_VEL
LIN {X 0,Y 91.765,Z 485.335,A -85,B 0,C 180,E1 -30227.522,E2 -30227.522} C_VEL
LIN {X 0,Y 103.474,Z 477.345,A -85,B 0,C 180,E1 -30229.98,E2 -30229.98} C_VEL
LIN {X 0,Y 115.307,Z 467.708,A -85,B 0,C 180,E1 -30232.036,E2 -30232.036} C_VEL
LIN {X 0,Y 125.705,Z 457.631,A -85,B 0,C 180,E1 -30233.58,E2 -30233.58} C_VEL
LIN {X 0,Y 135.848,Z 445.988,A -85,B 0,C 180,E1 -30234.754,E2 -30234.754} C_VEL
LIN {X 0,Y 144.464,Z 434.136,A -85,B 0,C 180,E1 -30235.735,E2 -30235.735} C_VEL
LIN {X 0,Y 152.254,Z 421.239,A -85,B 0,C 180,E1 -30236.501,E2 -30236.501} C_VEL
LIN {X 0,Y 159.172,Z 407.09,A -85,B 0,C 180,E1 -30237.276,E2 -30237.276} C_VEL
LIN {X 0,Y 164.627,Z 392.797,A -85,B 0,C 180,E1 -30237.896,E2 -30237.896} C_VEL
LIN {X 0,Y 168.734,Z 378.321,A -85,B 0,C 180,E1 -30238.315,E2 -30238.315} C_VEL
LIN {X 0,Y 171.561,Z 363.578,A -85,B 0,C 180,E1 -30238.655,E2 -30238.655} C_VEL
LIN {X 0,Y 173.874,Z 345.405,A -85,B 0,C 180,E1 -30238.985,E2 -30238.985} C_VEL
LIN {X 0,Y 173.861,Z 345.468,A -85,B 0,C 180,E1 -30239.927,E2 -30239.927} C_VEL
LIN {X 0,Y 170.694,Z 369.145,A -85,B 0,C 180,E1 -30240.278,E2 -30240.278} C_VEL
LIN {X 0,Y 167.204,Z 384.614,A -85,B 0,C 180,E1 -30240.498,E2 -30240.498} C_VEL
LIN {X 0,Y 162.467,Z 399.328,A -85,B 0,C 180,E1 -30240.701,E2 -30240.701} C_VEL
LIN {X 0,Y 156.386,Z 413.702,A -85,B 0,C 180,E1 -30240.991,E2 -30240.991} C_VEL
LIN {X 0,Y 149.374,Z 426.926,A -85,B 0,C 180,E1 -30241.319,E2 -30241.319} C_VEL
LIN {X 0,Y 140.619,Z 440.445,A -85,B 0,C 180,E1 -30241.796,E2 -30241.796} C_VEL
LIN {X 0,Y 131.003,Z 452.716,A -85,B 0,C 180,E1 -30242.415,E2 -30242.415} C_VEL
LIN {X 0,Y 120.699,Z 463.785,A -85,B 0,C 180,E1 -30243.338,E2 -30243.338} C_VEL
LIN {X 0,Y 112.745,Z 471.169,A -85,B 0,C 180,E1 -30244.231,E2 -30244.231} C_VEL
LIN {X 0,Y 100.646,Z 480.868,A -85,B 0,C 180,E1 -30245.754,E2 -30245.754} C_VEL
LIN {X 0,Y 88.68,Z 488.989,A -85,B 0,C 180,E1 -30247.891,E2 -30247.891} C_VEL
LIN {X 0,Y 74.97,Z 496.713,A -85,B 0,C 180,E1 -30251.242,E2 -30251.242} C_VEL
LIN {X 0,Y 62.165,Z 502.687,A -85,B 0,C 180,E1 -30256.093,E2 -30256.093} C_VEL
LIN {X 0,Y 49.793,Z 507.395,A -85,B 0,C 180,E1 -30263.474,E2 -30263.474} C_VEL
LIN {X 0,Y 41.358,Z 510.047,A -85,B 0,C 180,E1 -30271.85,E2 -30271.85} C_VEL
LIN {X 0,Y 32.252,Z 512.57,A -85,B 0,C 180,E1 -30289.199,E2 -30289.199} C_VEL
LIN {X 0,Y 27.888,Z 513.938,A -85,B 0,C 180,E1 -30315.423,E2 -30315.423} C_VEL
LIN {X 0,Y 28.12,Z 514.166,A -85,B 0,C 180,E1 -30331.467,E2 -30331.467} C_VEL
LIN {X 0,Y 29.334,Z 513.38,A -85,B 0,C 180,E1 -30358.65,E2 -30358.65} C_VEL
LIN {X 0,Y 36.42,Z 511.41,A -85,B 0,C 180,E1 -30380.545,E2 -30380.545} C_VEL
LIN {X 0,Y 48.695,Z 507.671,A -85,B 0,C 180,E1 -30395.621,E2 -30395.621} C_VEL
LIN {X 0,Y 49.978,Z 507.031,A -85,B 0,C 180,E1 -30398.039,E2 -30398.039} C_VEL
LIN {X 0,Y 50.671,Z 503.752,A -85,B 0,C 180,E1 -30427.973,E2 -30427.973} C_VEL
LIN {X 0,Y 58.165,Z 501.46,A -85,B 0,C 180,E1 -30443.498,E2 -30443.498} C_VEL
LIN {X 0,Y 55.327,Z 502.536,A -85,B 0,C 180,E1 -30447.21,E2 -30447.21} C_VEL
LIN {X 0,Y 44.199,Z 505.963,A -85,B 0,C 180,E1 -30457.323,E2 -30457.323} C_VEL
LIN {X 0,Y 34.426,Z 508.332,A -85,B 0,C 180,E1 -30474.747,E2 -30474.747} C_VEL
LIN {X 0,Y 29.773,Z 509.268,A -85,B 0,C 180,E1 -30494.407,E2 -30494.407} C_VEL
LIN {X 0,Y 28.206,Z 509.569,A -85,B 0,C 180,E1 -30505.659,E2 -30505.659} C_VEL
LIN {X 0,Y 26.229,Z 509.717,A -85,B 0,C 180,E1 -30526.234,E2 -30526.234} C_VEL
LIN {X 0,Y 26.926,Z 509.411,A -85,B 0,C 180,E1 -30543.49,E2 -30543.49} C_VEL
LIN {X 0,Y 29.467,Z 508.868,A -85,B 0,C 180,E1 -30554.434,E2 -30554.434} C_VEL
LIN {X 0,Y 30.707,Z 508.619,A -85,B 0,C 180,E1 -30557.357,E2 -30557.357} C_VEL
LIN {X 0,Y 40.259,Z 506.623,A -85,B 0,C 180,E1 -30570.765,E2 -30570.765} C_VEL
LIN {X 0,Y 52.425,Z 503.238,A -85,B 0,C 180,E1 -30579.755,E2 -30579.755} C_VEL
LIN {X 0,Y 65.317,Z 498.581,A -85,B 0,C 180,E1 -30585.521,E2 -30585.521} C_VEL
LIN {X 0,Y 78.646,Z 492.5,A -85,B 0,C 180,E1 -30589.379,E2 -30589.379} C_VEL
LIN {X 0,Y 92.204,Z 484.832,A -85,B 0,C 180,E1 -30592.215,E2 -30592.215} C_VEL
LIN {X 0,Y 104.205,Z 476.621,A -85,B 0,C 180,E1 -30594.102,E2 -30594.102} C_VEL
LIN {X 0,Y 116.271,Z 466.713,A -85,B 0,C 180,E1 -30595.752,E2 -30595.752} C_VEL
LIN {X 0,Y 126.671,Z 456.561,A -85,B 0,C 180,E1 -30596.973,E2 -30596.973} C_VEL
LIN {X 0,Y 136.256,Z 445.477,A -85,B 0,C 180,E1 -30597.822,E2 -30597.822} C_VEL
LIN {X 0,Y 140.619,Z 439.734,A -85,B 0,C 180,E1 -30598.204,E2 -30598.204} C_VEL
LIN {X 0,Y 140.576,Z 439.872,A -85,B 0,C 180,E1 -30598.899,E2 -30598.899} C_VEL
LIN {X 0,Y 130.896,Z 452.138,A -85,B 0,C 180,E1 -30599.299,E2 -30599.299} C_VEL
LIN {X 0,Y 121.046,Z 462.644,A -85,B 0,C 180,E1 -30599.908,E2 -30599.908} C_VEL
LIN {X 0,Y 112.444,Z 470.587,A -85,B 0,C 180,E1 -30600.611,E2 -30600.611} C_VEL
LIN {X 0,Y 100.182,Z 480.281,A -85,B 0,C 180,E1 -30601.677,E2 -30601.677} C_VEL
LIN {X 0,Y 87.982,Z 488.399,A -85,B 0,C 180,E1 -30603.252,E2 -30603.252} C_VEL
LIN {X 0,Y 76.111,Z 495.042,A -85,B 0,C 180,E1 -30605.298,E2 -30605.298} C_VEL
LIN {X 0,Y 63.93,Z 500.696,A -85,B 0,C 180,E1 -30608.41,E2 -30608.41} C_VEL
LIN {X 0,Y 50.625,Z 505.722,A -85,B 0,C 180,E1 -30613.69,E2 -30613.69} C_VEL
LIN {X 0,Y 38.048,Z 509.452,A -85,B 0,C 180,E1 -30622.584,E2 -30622.584} C_VEL
LIN {X 0,Y 27.211,Z 511.975,A -85,B 0,C 180,E1 -30639.239,E2 -30639.239} C_VEL
LIN {X 0,Y 21.01,Z 513.344,A -85,B 0,C 180,E1 -30670.484,E2 -30670.484} C_VEL
LIN {X 0,Y 21.042,Z 513.595,A -85,B 0,C 180,E1 -30690.024,E2 -30690.024} C_VEL
LIN {X 0,Y 23.285,Z 512.786,A -85,B 0,C 180,E1 -30727.158,E2 -30727.158} C_VEL
LIN {X 0,Y 32.324,Z 510.814,A -85,B 0,C 180,E1 -30750.454,E2 -30750.454} C_VEL
LIN {X 0,Y 40.68,Z 508.718,A -85,B 0,C 180,E1 -30759.787,E2 -30759.787} C_VEL
LIN {X 0,Y 42.09,Z 508.062,A -85,B 0,C 180,E1 -30763.011,E2 -30763.011} C_VEL
LIN {X 0,Y 46.706,Z 504.799,A -85,B 0,C 180,E1 -30797.515,E2 -30797.515} C_VEL
LIN {X 0,Y 48.575,Z 504.322,A -85,B 0,C 180,E1 -30801.345,E2 -30801.345} C_VEL
LIN {X 0,Y 47.482,Z 504.645,A -85,B 0,C 180,E1 -30803.364,E2 -30803.364} C_VEL
LIN {X 0,Y 34.711,Z 507.814,A -85,B 0,C 180,E1 -30815.89,E2 -30815.89} C_VEL
LIN {X 0,Y 25.621,Z 509.481,A -85,B 0,C 180,E1 -30836.704,E2 -30836.704} C_VEL
LIN {X 0,Y 21.731,Z 510.06,A -85,B 0,C 180,E1 -30869.976,E2 -30869.976} C_VEL
LIN {X 0,Y 25.608,Z 509.504,A -85,B 0,C 180,E1 -30903.267,E2 -30903.267} C_VEL
LIN {X 0,Y 30.707,Z 508.619,A -85,B 0,C 180,E1 -30917.357,E2 -30917.357} C_VEL
LIN {X 0,Y 34.465,Z 507.902,A -85,B 0,C 180,E1 -30925.263,E2 -30925.263} C_VEL
LIN {X 0,Y 40.629,Z 506.471,A -85,B 0,C 180,E1 -30936.973,E2 -30936.973} C_VEL
LIN {X 0,Y 46.311,Z 504.998,A -85,B 0,C 180,E1 -30944.094,E2 -30944.094} C_VEL
LIN {X 0,Y 51.241,Z 503.573,A -85,B 0,C 180,E1 -30947.604,E2 -30947.604} C_VEL
LIN {X 0,Y 53.013,Z 503.03,A -85,B 0,C 180,E1 -30948.375,E2 -30948.375} C_VEL
LIN {X 0,Y 63.916,Z 499.164,A -85,B 0,C 180,E1 -30951.677,E2 -30951.677} C_VEL
LIN {X 0,Y 77.65,Z 493.085,A -85,B 0,C 180,E1 -30954.544,E2 -30954.544} C_VEL
LIN {X 0,Y 91.514,Z 485.413,A -85,B 0,C 180,E1 -30956.616,E2 -30956.616} C_VEL
LIN {X 0,Y 98.48,Z 480.901,A -85,B 0,C 180,E1 -30957.446,E2 -30957.446} C_VEL
LIN {X 0,Y 98.462,Z 480.935,A -85,B 0,C 180,E1 -30957.69,E2 -30957.69} C_VEL
LIN {X 0,Y 86.104,Z 488.832,A -85,B 0,C 180,E1 -30958.734,E2 -30958.734} C_VEL
LIN {X 0,Y 73.427,Z 495.577,A -85,B 0,C 180,E1 -30960.178,E2 -30960.178} C_VEL
LIN {X 0,Y 59.794,Z 501.498,A -85,B 0,C 180,E1 -30962.684,E2 -30962.684} C_VEL
LIN {X 0,Y 45.996,Z 506.208,A -85,B 0,C 180,E1 -30966.794,E2 -30966.794} C_VEL
LIN {X 0,Y 35.898,Z 508.855,A -85,B 0,C 180,E1 -30971.869,E2 -30971.869} C_VEL
LIN {X 0,Y 23.331,Z 511.38,A -85,B 0,C 180,E1 -30985.406,E2 -30985.406} C_VEL
LIN {X 0,Y 14.442,Z 512.75,A -85,B 0,C 180,E1 -31020.921,E2 -31020.921} C_VEL
LIN {X 0,Y 13.855,Z 513.001,A -85,B 0,C 180,E1 -31050.037,E2 -31050.037} C_VEL
LIN {X 0,Y 18.069,Z 512.189,A -85,B 0,C 180,E1 -31101.115,E2 -31101.115} C_VEL
LIN {X 0,Y 29.443,Z 510.218,A -85,B 0,C 180,E1 -31122.764,E2 -31122.764} C_VEL
LIN {X 0,Y 34.719,Z 508.996,A -85,B 0,C 180,E1 -31128.323,E2 -31128.323} C_VEL
LIN {X 0,Y 38.662,Z 506.871,A -85,B 0,C 180,E1 -31156.885,E2 -31156.885} C_VEL
LIN {X 0,Y 37.349,Z 507.135,A -85,B 0,C 180,E1 -31159.764,E2 -31159.764} C_VEL
LIN {X 0,Y 25.231,Z 509.374,A -85,B 0,C 180,E1 -31173.28,E2 -31173.28} C_VEL
LIN {X 0,Y 16.205,Z 510.494,A -85,B 0,C 180,E1 -31204.263,E2 -31204.263} C_VEL
LIN {X 0,Y 16.195,Z 510.501,A -85,B 0,C 180,E1 -31255.683,E2 -31255.683} C_VEL
LIN {X 0,Y 25.215,Z 509.41,A -85,B 0,C 180,E1 -31286.698,E2 -31286.698} C_VEL
LIN {X 0,Y 37.311,Z 507.209,A -85,B 0,C 180,E1 -31300.318,E2 -31300.318} C_VEL
LIN {X 0,Y 50.408,Z 503.824,A -85,B 0,C 180,E1 -31307.361,E2 -31307.361} C_VEL
LIN {X 0,Y 53.013,Z 503.03,A -85,B 0,C 180,E1 -31308.375,E2 -31308.375} C_VEL
LIN {X 0,Y 53.083,Z 503.039,A -85,B 0,C 180,E1 -31309.345,E2 -31309.345} C_VEL
LIN {X 0,Y 51.495,Z 503.606,A -85,B 0,C 180,E1 -31311.228,E2 -31311.228} C_VEL
LIN {X 0,Y 46.591,Z 505.19,A -85,B 0,C 180,E1 -31314.112,E2 -31314.112} C_VEL
LIN {X 0,Y 35.136,Z 508.198,A -85,B 0,C 180,E1 -31319.058,E2 -31319.058} C_VEL
LIN {X 0,Y 29.74,Z 509.371,A -85,B 0,C 180,E1 -31321.923,E2 -31321.923} C_VEL
LIN {X 0,Y 24.298,Z 510.291,A -85,B 0,C 180,E1 -31325.275,E2 -31325.275} C_VEL
LIN {X 0,Y 14.644,Z 511.615,A -85,B 0,C 180,E1 -31336.418,E2 -31336.418} C_VEL
LIN {X 0,Y 6.681,Z 512.408,A -85,B 0,C 180,E1 -31410.077,E2 -31410.077} C_VEL
LIN {X 0,Y 14.662,Z 511.594,A -85,B 0,C 180,E1 -31483.592,E2 -31483.592} C_VEL
LIN {X 0,Y 21.279,Z 510.751,A -85,B 0,C 180,E1 -31492.408,E2 -31492.408} C_VEL
LIN {X 0,Y 28.002,Z 509.515,A -85,B 0,C 180,E1 -31500.002,E2 -31500.002} C_VEL
